KUKA KRL program: EPS_2_26115_SA7006_A_20260219035544.src

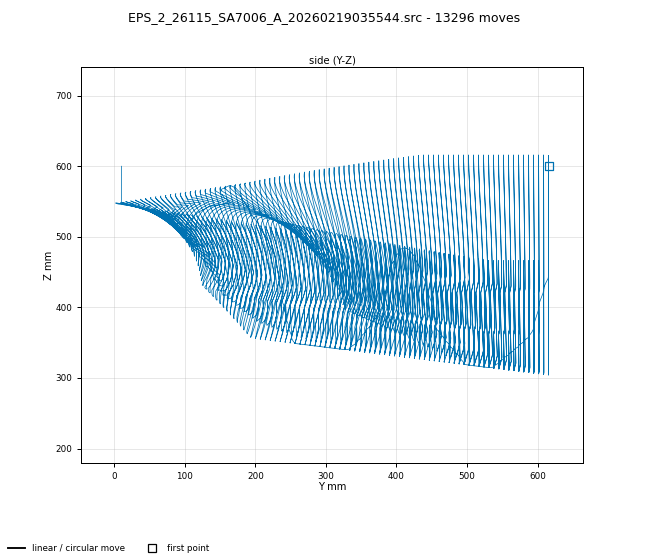
[picture p0: tool path of EPS_2_26115_SA7006_A_20260219035544.src, 13296 of 13298 moves have a stored position in this frame; points joined in program order, loops and branches not executed]
&ACCESS RVP
&REL 4
&COMMENT QRS 19112012
&PARAM EDITMASK = *
DEF PART()
EXT BAS (BAS_COMMAND :IN,REAL :IN )
INT I
BAS (#INITMOV,0 )

;KUKA QRS Post kuka4.cps  Date:22-06-2017 !

File_ID=3062

QRS_PRE_INIT()

;Init var - Until changes are made in qrs_pre_init
Outlet_Square_prg=0
Inlet_1_Square_prg=0
Inlet_2_Square_prg=0
Inlet_3_Square_prg=0
Inlet_4_Square_prg=0
Inlet_5_Square_prg=0

Outlet_1={X 0.000, Y 435.000, Z 433.000, B 0.000, E1 0.000 }
Inlet_1={X 0.000, Y 529.410, Z 340.500, B 0.000, E1 90.000 }
Inlet_2={X 0.000, Y 529.410, Z 340.500, B 0.000, E1 180.000 }
Outlet_1_type=366
Inlet_1_type=201
Inlet_2_type=201
;QRS#1=Sidecore dimensions
;QRS#2=375-15" PVC SDR 35 Cut Back
;QRS#3=200-8" PVC SDR 35
;QRS#4=200-8" PVC SDR 35
;QRS#5=
;QRS#6=
;QRS#7=
;QRS#8=
;QRS#9=20Y PSX
;QRS#10=12-08 PSX
;QRS#11=12-08 PSX
;QRS#12=
;QRS#13=
;QRS#14=
;QRS#15=
;QRS#16=1220x127x914 3'
;QRS#17=EPS Height
;QRS#18=616
;QRS#19=*
;QRS#20= UPDATED VERSION 22-06-2017
;QRS#21=*
Outlet_Square=0250
Inlet_1_Square=0100
Inlet_2_Square=0100
Inlet_3_Square=0
Inlet_4_Square=0
Inlet_5_Square=0
Mill_Square=1
Outlet_Square_Prg=275
Inlet_1_Square_prg=204
Inlet_2_Square_prg=204

QRS_INIT()

$ADVANCE=5

; T1
PTP {E1 173.498,E2 173.498}
PTP {X 0,Y 615.498,A -85,B 0,C 180,E1 173.498,E2 173.498,E3 0,E4 0,E5 0,E6 0}
QRS_SPEED_INIT()
LIN {X 0,Y 615.498,Z 600,A -85,B 0,C 180,E1 173.498,E2 173.498,E3 0,E4 0,E5 0,E6 0} C_VEL
LIN {X 0,Y 615.498,Z 456.733,A -85,B 0,C 180,E1 173.498,E2 173.498} C_VEL
LIN {X 0,Y 615.498,Z 445.854,A -85,B 0,C 180,E1 173.498,E2 173.498} C_VEL
LIN {X 0,Y 615.496,Z 444.21,A -85,B 0,C 180,E1 173.418,E2 173.418} C_VEL
LIN {X 0,Y 615.497,Z 436.534,A -85,B 0,C 180,E1 172.454,E2 172.454} C_VEL
LIN {X 0,Y 615.498,Z 426.756,A -85,B 0,C 180,E1 171.463,E2 171.463} C_VEL
LIN {X 0,Y 615.498,Z 416.489,A -85,B 0,C 180,E1 170.635,E2 170.635} C_VEL
LIN {X 0,Y 615.464,Z 404.93,A -85,B 0,C 180,E1 169.888,E2 169.888} C_VEL
LIN {X 0,Y 615.482,Z 393.083,A -85,B 0,C 180,E1 169.293,E2 169.293} C_VEL
LIN {X 0,Y 615.493,Z 380.15,A -85,B 0,C 180,E1 168.807,E2 168.807} C_VEL
LIN {X 0,Y 615.483,Z 367.548,A -85,B 0,C 180,E1 168.473,E2 168.473} C_VEL
LIN {X 0,Y 615.474,Z 360.281,A -85,B 0,C 180,E1 168.327,E2 168.327} C_VEL
LIN {X 0,Y 615.446,Z 354.613,A -85,B 0,C 180,E1 166.085,E2 166.085} C_VEL
LIN {X 0,Y 615.469,Z 347.897,A -85,B 0,C 180,E1 163.413,E2 163.413} C_VEL
LIN {X 0,Y 615.435,Z 341.109,A -85,B 0,C 180,E1 160.66,E2 160.66} C_VEL
LIN {X 0,Y 615.436,Z 335.997,A -85,B 0,C 180,E1 158.566,E2 158.566} C_VEL
LIN {X 0,Y 615.464,Z 329.821,A -85,B 0,C 180,E1 155.998,E2 155.998} C_VEL
LIN {X 0,Y 615.491,Z 324.07,A -85,B 0,C 180,E1 153.556,E2 153.556} C_VEL
LIN {X 0,Y 615.488,Z 318.958,A -85,B 0,C 180,E1 151.342,E2 151.342} C_VEL
LIN {X 0,Y 615.493,Z 313.469,A -85,B 0,C 180,E1 148.914,E2 148.914} C_VEL
LIN {X 0,Y 615.495,Z 307.987,A -85,B 0,C 180,E1 146.466,E2 146.466} C_VEL
LIN {X 0,Y 615.477,Z 304.012,A -85,B 0,C 180,E1 144.684,E2 144.684} C_VEL
LIN {X 0,Y 615.479,Z 304.01,A -85,B 0,C 180,E1 141.93,E2 141.93} C_VEL
LIN {X 0,Y 615.492,Z 304.007,A -85,B 0,C 180,E1 139.394,E2 139.394} C_VEL
LIN {X 0,Y 615.463,Z 304.012,A -85,B 0,C 180,E1 136.753,E2 136.753} C_VEL
LIN {X 0,Y 615.466,Z 304.012,A -85,B 0,C 180,E1 133.995,E2 133.995} C_VEL
LIN {X 0,Y 615.494,Z 304.011,A -85,B 0,C 180,E1 131.095,E2 131.095} C_VEL
LIN {X 0,Y 615.469,Z 304.011,A -85,B 0,C 180,E1 128.907,E2 128.907} C_VEL
LIN {X 0,Y 615.462,Z 304.013,A -85,B 0,C 180,E1 126.428,E2 126.428} C_VEL
LIN {X 0,Y 615.481,Z 304.167,A -85,B 0,C 180,E1 124.817,E2 124.817} C_VEL
LIN {X 0,Y 615.49,Z 310.295,A -85,B 0,C 180,E1 122.331,E2 122.331} C_VEL
LIN {X 0,Y 615.491,Z 316.167,A -85,B 0,C 180,E1 119.795,E2 119.795} C_VEL
LIN {X 0,Y 615.44,Z 322.494,A -85,B 0,C 180,E1 117.036,E2 117.036} C_VEL
LIN {X 0,Y 615.448,Z 327.267,A -85,B 0,C 180,E1 114.995,E2 114.995} C_VEL
LIN {X 0,Y 615.492,Z 333.562,A -85,B 0,C 180,E1 112.346,E2 112.346} C_VEL
LIN {X 0,Y 615.488,Z 339.166,A -85,B 0,C 180,E1 110.034,E2 110.034} C_VEL
LIN {X 0,Y 615.48,Z 345.979,A -85,B 0,C 180,E1 107.272,E2 107.272} C_VEL
LIN {X 0,Y 615.469,Z 352.77,A -85,B 0,C 180,E1 104.551,E2 104.551} C_VEL
LIN {X 0,Y 615.487,Z 359.577,A -85,B 0,C 180,E1 101.862,E2 101.862} C_VEL
LIN {X 0,Y 615.494,Z 360.311,A -85,B 0,C 180,E1 101.57,E2 101.57} C_VEL
LIN {X 0,Y 615.491,Z 372.644,A -85,B 0,C 180,E1 101.319,E2 101.319} C_VEL
LIN {X 0,Y 615.456,Z 385.792,A -85,B 0,C 180,E1 100.911,E2 100.911} C_VEL
LIN {X 0,Y 615.455,Z 398.542,A -85,B 0,C 180,E1 100.363,E2 100.363} C_VEL
LIN {X 0,Y 615.497,Z 410.282,A -85,B 0,C 180,E1 99.697,E2 99.697} C_VEL
LIN {X 0,Y 615.499,Z 420.75,A -85,B 0,C 180,E1 98.952,E2 98.952} C_VEL
LIN {X 0,Y 615.498,Z 429.315,A -85,B 0,C 180,E1 98.207,E2 98.207} C_VEL
LIN {X 0,Y 615.497,Z 437.196,A -85,B 0,C 180,E1 97.382,E2 97.382} C_VEL
LIN {X 0,Y 615.497,Z 444.889,A -85,B 0,C 180,E1 96.393,E2 96.393} C_VEL
LIN {X 0,Y 615.497,Z 451.95,A -85,B 0,C 180,E1 95.243,E2 95.243} C_VEL
LIN {X 0,Y 615.494,Z 456.651,A -85,B 0,C 180,E1 94.258,E2 94.258} C_VEL
LIN {X 0,Y 615.494,Z 460.25,A -85,B 0,C 180,E1 93.274,E2 93.274} C_VEL
LIN {X 0,Y 615.496,Z 462.111,A -85,B 0,C 180,E1 92.619,E2 92.619} C_VEL
LIN {X 0,Y 615.499,Z 463.53,A -85,B 0,C 180,E1 91.965,E2 91.965} C_VEL
LIN {X 0,Y 615.496,Z 465.14,A -85,B 0,C 180,E1 90.656,E2 90.656} C_VEL
LIN {X 0,Y 615.495,Z 465.384,A -85,B 0,C 180,E1 90.002,E2 90.002} C_VEL
LIN {X 0,Y 615.495,Z 465.207,A -85,B 0,C 180,E1 89.347,E2 89.347} C_VEL
LIN {X 0,Y 615.499,Z 463.685,A -85,B 0,C 180,E1 88.039,E2 88.039} C_VEL
LIN {X 0,Y 615.498,Z 462.345,A -85,B 0,C 180,E1 87.384,E2 87.384} C_VEL
LIN {X 0,Y 615.496,Z 459.499,A -85,B 0,C 180,E1 86.401,E2 86.401} C_VEL
LIN {X 0,Y 615.498,Z 455.641,A -85,B 0,C 180,E1 85.417,E2 85.417} C_VEL
LIN {X 0,Y 615.498,Z 450.661,A -85,B 0,C 180,E1 84.432,E2 84.432} C_VEL
LIN {X 0,Y 615.496,Z 444.209,A -85,B 0,C 180,E1 83.418,E2 83.418} C_VEL
LIN {X 0,Y 615.497,Z 436.553,A -85,B 0,C 180,E1 82.456,E2 82.456} C_VEL
LIN {X 0,Y 615.498,Z 426.778,A -85,B 0,C 180,E1 81.465,E2 81.465} C_VEL
LIN {X 0,Y 615.498,Z 416.518,A -85,B 0,C 180,E1 80.637,E2 80.637} C_VEL
LIN {X 0,Y 615.472,Z 404.964,A -85,B 0,C 180,E1 79.89,E2 79.89} C_VEL
LIN {X 0,Y 615.444,Z 393.348,A -85,B 0,C 180,E1 79.303,E2 79.303} C_VEL
LIN {X 0,Y 615.466,Z 381.479,A -85,B 0,C 180,E1 78.849,E2 78.849} C_VEL
LIN {X 0,Y 615.491,Z 369.465,A -85,B 0,C 180,E1 78.517,E2 78.517} C_VEL
LIN {X 0,Y 615.495,Z 360.283,A -85,B 0,C 180,E1 78.329,E2 78.329} C_VEL
LIN {X 0,Y 615.49,Z 354.559,A -85,B 0,C 180,E1 76.068,E2 76.068} C_VEL
LIN {X 0,Y 615.472,Z 347.903,A -85,B 0,C 180,E1 73.415,E2 73.415} C_VEL
LIN {X 0,Y 615.476,Z 341.109,A -85,B 0,C 180,E1 70.664,E2 70.664} C_VEL
LIN {X 0,Y 615.488,Z 334.288,A -85,B 0,C 180,E1 67.866,E2 67.866} C_VEL
LIN {X 0,Y 615.489,Z 329.182,A -85,B 0,C 180,E1 65.73,E2 65.73} C_VEL
LIN {X 0,Y 615.467,Z 324.079,A -85,B 0,C 180,E1 63.557,E2 63.557} C_VEL
LIN {X 0,Y 615.437,Z 318.971,A -85,B 0,C 180,E1 61.342,E2 61.342} C_VEL
LIN {X 0,Y 615.489,Z 313.418,A -85,B 0,C 180,E1 58.914,E2 58.914} C_VEL
LIN {X 0,Y 615.499,Z 307.609,A -85,B 0,C 180,E1 56.465,E2 56.465} C_VEL
LIN {X 0,Y 615.481,Z 304.007,A -85,B 0,C 180,E1 54.988,E2 54.988} C_VEL
LIN {X 0,Y 615.475,Z 304.002,A -85,B 0,C 180,E1 52.76,E2 52.76} C_VEL
LIN {X 0,Y 615.48,Z 304.012,A -85,B 0,C 180,E1 49.912,E2 49.912} C_VEL
LIN {X 0,Y 615.433,Z 304.012,A -85,B 0,C 180,E1 47.646,E2 47.646} C_VEL
LIN {X 0,Y 615.48,Z 304.013,A -85,B 0,C 180,E1 44.934,E2 44.934} C_VEL
LIN {X 0,Y 615.468,Z 304.004,A -85,B 0,C 180,E1 42.082,E2 42.082} C_VEL
LIN {X 0,Y 615.487,Z 304.01,A -85,B 0,C 180,E1 39.751,E2 39.751} C_VEL
LIN {X 0,Y 615.471,Z 304.003,A -85,B 0,C 180,E1 36.939,E2 36.939} C_VEL
LIN {X 0,Y 615.46,Z 304.012,A -85,B 0,C 180,E1 34.024,E2 34.024} C_VEL
LIN {X 0,Y 615.429,Z 304.012,A -85,B 0,C 180,E1 31.689,E2 31.689} C_VEL
LIN {X 0,Y 615.463,Z 304.012,A -85,B 0,C 180,E1 29.408,E2 29.408} C_VEL
LIN {X 0,Y 615.477,Z 304.002,A -85,B 0,C 180,E1 26.445,E2 26.445} C_VEL
LIN {X 0,Y 615.483,Z 304.011,A -85,B 0,C 180,E1 24.014,E2 24.014} C_VEL
LIN {X 0,Y 615.458,Z 304.007,A -85,B 0,C 180,E1 21.433,E2 21.433} C_VEL
LIN {X 0,Y 615.49,Z 304.015,A -85,B 0,C 180,E1 18.614,E2 18.614} C_VEL
LIN {X 0,Y 615.432,Z 304.012,A -85,B 0,C 180,E1 15.907,E2 15.907} C_VEL
LIN {X 0,Y 615.495,Z 304.008,A -85,B 0,C 180,E1 13.201,E2 13.201} C_VEL
LIN {X 0,Y 615.477,Z 304.003,A -85,B 0,C 180,E1 10.527,E2 10.527} C_VEL
LIN {X 0,Y 615.478,Z 304.01,A -85,B 0,C 180,E1 7.876,E2 7.876} C_VEL
LIN {X 0,Y 615.469,Z 304.005,A -85,B 0,C 180,E1 5.242,E2 5.242} C_VEL
LIN {X 0,Y 615.463,Z 304.012,A -85,B 0,C 180,E1 2.618,E2 2.618} C_VEL
LIN {X 0,Y 615.444,Z 304.011,A -85,B 0,C 180,E1 0,E2 0} C_VEL
LIN {X 0,Y 615.491,Z 304.006,A -85,B 0,C 180,E1 -2.618,E2 -2.618} C_VEL
LIN {X 0,Y 615.481,Z 304.002,A -85,B 0,C 180,E1 -5.241,E2 -5.241} C_VEL
LIN {X 0,Y 615.473,Z 304.01,A -85,B 0,C 180,E1 -7.876,E2 -7.876} C_VEL
LIN {X 0,Y 615.461,Z 304.007,A -85,B 0,C 180,E1 -10.527,E2 -10.527} C_VEL
LIN {X 0,Y 615.456,Z 304.012,A -85,B 0,C 180,E1 -13.202,E2 -13.202} C_VEL
LIN {X 0,Y 615.46,Z 304.007,A -85,B 0,C 180,E1 -15.226,E2 -15.226} C_VEL
LIN {X 0,Y 615.484,Z 304.012,A -85,B 0,C 180,E1 -17.957,E2 -17.957} C_VEL
LIN {X 0,Y 615.492,Z 303.998,A -85,B 0,C 180,E1 -20.73,E2 -20.73} C_VEL
LIN {X 0,Y 615.474,Z 304.011,A -85,B 0,C 180,E1 -23.557,E2 -23.557} C_VEL
LIN {X 0,Y 615.437,Z 304.012,A -85,B 0,C 180,E1 -25.718,E2 -25.718} C_VEL
LIN {X 0,Y 615.481,Z 304.013,A -85,B 0,C 180,E1 -28.455,E2 -28.455} C_VEL
LIN {X 0,Y 615.462,Z 304.005,A -85,B 0,C 180,E1 -31.087,E2 -31.087} C_VEL
LIN {X 0,Y 615.478,Z 304.009,A -85,B 0,C 180,E1 -33.538,E2 -33.538} C_VEL
LIN {X 0,Y 615.481,Z 304.001,A -85,B 0,C 180,E1 -36.425,E2 -36.425} C_VEL
LIN {X 0,Y 615.492,Z 304.014,A -85,B 0,C 180,E1 -39.067,E2 -39.067} C_VEL
LIN {X 0,Y 615.433,Z 304.012,A -85,B 0,C 180,E1 -41.478,E2 -41.478} C_VEL
LIN {X 0,Y 615.48,Z 304.013,A -85,B 0,C 180,E1 -44.15,E2 -44.15} C_VEL
LIN {X 0,Y 615.464,Z 304.005,A -85,B 0,C 180,E1 -46.955,E2 -46.955} C_VEL
LIN {X 0,Y 615.489,Z 304.011,A -85,B 0,C 180,E1 -49.397,E2 -49.397} C_VEL
LIN {X 0,Y 615.471,Z 304.003,A -85,B 0,C 180,E1 -51.99,E2 -51.99} C_VEL
LIN {X 0,Y 615.497,Z 304.002,A -85,B 0,C 180,E1 -54.388,E2 -54.388} C_VEL
LIN {X 0,Y 615.444,Z 304.194,A -85,B 0,C 180,E1 -55.768,E2 -55.768} C_VEL
LIN {X 0,Y 615.497,Z 324.712,A -85,B 0,C 180,E1 -58.468,E2 -58.468} C_VEL
LIN {X 0,Y 615.482,Z 347.265,A -85,B 0,C 180,E1 -61.344,E2 -61.344} C_VEL
LIN {X 0,Y 615.489,Z 369.495,A -85,B 0,C 180,E1 -64.105,E2 -64.105} C_VEL
LIN {X 0,Y 615.479,Z 391.725,A -85,B 0,C 180,E1 -66.802,E2 -66.802} C_VEL
LIN {X 0,Y 615.491,Z 415.039,A -85,B 0,C 180,E1 -69.574,E2 -69.574} C_VEL
LIN {X 0,Y 615.494,Z 421.023,A -85,B 0,C 180,E1 -70.252,E2 -70.252} C_VEL
LIN {X 0,Y 615.487,Z 444.892,A -85,B 0,C 180,E1 -70.578,E2 -70.578} C_VEL
LIN {X 0,Y 615.475,Z 460.906,A -85,B 0,C 180,E1 -70.924,E2 -70.924} C_VEL
LIN {X 0,Y 615.493,Z 476.391,A -85,B 0,C 180,E1 -71.393,E2 -71.393} C_VEL
LIN {X 0,Y 615.488,Z 491.252,A -85,B 0,C 180,E1 -71.964,E2 -71.964} C_VEL
LIN {X 0,Y 615.499,Z 505.771,A -85,B 0,C 180,E1 -72.646,E2 -72.646} C_VEL
LIN {X 0,Y 615.498,Z 520.515,A -85,B 0,C 180,E1 -73.49,E2 -73.49} C_VEL
LIN {X 0,Y 615.497,Z 534.385,A -85,B 0,C 180,E1 -74.437,E2 -74.437} C_VEL
LIN {X 0,Y 615.495,Z 547.051,A -85,B 0,C 180,E1 -75.453,E2 -75.453} C_VEL
LIN {X 0,Y 615.493,Z 559.563,A -85,B 0,C 180,E1 -76.633,E2 -76.633} C_VEL
LIN {X 0,Y 615.49,Z 570.189,A -85,B 0,C 180,E1 -77.807,E2 -77.807} C_VEL
LIN {X 0,Y 615.49,Z 580.236,A -85,B 0,C 180,E1 -79.11,E2 -79.11} C_VEL
LIN {X 0,Y 615.495,Z 588.995,A -85,B 0,C 180,E1 -80.472,E2 -80.472} C_VEL
LIN {X 0,Y 615.495,Z 596.117,A -85,B 0,C 180,E1 -81.796,E2 -81.796} C_VEL
LIN {X 0,Y 615.491,Z 601.986,A -85,B 0,C 180,E1 -83.103,E2 -83.103} C_VEL
LIN {X 0,Y 615.492,Z 607.746,A -85,B 0,C 180,E1 -84.761,E2 -84.761} C_VEL
LIN {X 0,Y 615.493,Z 611.08,A -85,B 0,C 180,E1 -86.073,E2 -86.073} C_VEL
LIN {X 0,Y 615.485,Z 613.507,A -85,B 0,C 180,E1 -87.384,E2 -87.384} C_VEL
LIN {X 0,Y 615.488,Z 614.871,A -85,B 0,C 180,E1 -88.693,E2 -88.693} C_VEL
LIN {X 0,Y 615.489,Z 615.39,A -85,B 0,C 180,E1 -90.002,E2 -90.002} C_VEL
LIN {X 0,Y 615.488,Z 614.869,A -85,B 0,C 180,E1 -91.31,E2 -91.31} C_VEL
LIN {X 0,Y 615.485,Z 613.502,A -85,B 0,C 180,E1 -92.619,E2 -92.619} C_VEL
LIN {X 0,Y 615.493,Z 611.073,A -85,B 0,C 180,E1 -93.93,E2 -93.93} C_VEL
LIN {X 0,Y 615.492,Z 607.736,A -85,B 0,C 180,E1 -95.243,E2 -95.243} C_VEL
LIN {X 0,Y 615.492,Z 601.979,A -85,B 0,C 180,E1 -96.899,E2 -96.899} C_VEL
LIN {X 0,Y 615.489,Z 594.494,A -85,B 0,C 180,E1 -98.538,E2 -98.538} C_VEL
LIN {X 0,Y 615.496,Z 585.955,A -85,B 0,C 180,E1 -100.029,E2 -100.029} C_VEL
LIN {X 0,Y 615.494,Z 576.756,A -85,B 0,C 180,E1 -101.361,E2 -101.361} C_VEL
LIN {X 0,Y 615.495,Z 567.279,A -85,B 0,C 180,E1 -102.531,E2 -102.531} C_VEL
LIN {X 0,Y 615.496,Z 556.199,A -85,B 0,C 180,E1 -103.707,E2 -103.707} C_VEL
LIN {X 0,Y 615.495,Z 544.099,A -85,B 0,C 180,E1 -104.804,E2 -104.804} C_VEL
LIN {X 0,Y 615.497,Z 529.69,A -85,B 0,C 180,E1 -105.906,E2 -105.906} C_VEL
LIN {X 0,Y 615.497,Z 514.993,A -85,B 0,C 180,E1 -106.844,E2 -106.844} C_VEL
LIN {X 0,Y 615.499,Z 500.484,A -85,B 0,C 180,E1 -107.614,E2 -107.614} C_VEL
LIN {X 0,Y 615.486,Z 485.241,A -85,B 0,C 180,E1 -108.282,E2 -108.282} C_VEL
LIN {X 0,Y 615.48,Z 469.949,A -85,B 0,C 180,E1 -108.82,E2 -108.82} C_VEL
LIN {X 0,Y 615.478,Z 453.466,A -85,B 0,C 180,E1 -109.253,E2 -109.253} C_VEL
LIN {X 0,Y 615.494,Z 437.841,A -85,B 0,C 180,E1 -109.534,E2 -109.534} C_VEL
LIN {X 0,Y 615.494,Z 420.778,A -85,B 0,C 180,E1 -109.751,E2 -109.751} C_VEL
LIN {X 0,Y 615.496,Z 396.751,A -85,B 0,C 180,E1 -112.595,E2 -112.595} C_VEL
LIN {X 0,Y 615.489,Z 373.317,A -85,B 0,C 180,E1 -115.427,E2 -115.427} C_VEL
LIN {X 0,Y 615.488,Z 349.955,A -85,B 0,C 180,E1 -118.318,E2 -118.318} C_VEL
LIN {X 0,Y 615.474,Z 328.189,A -85,B 0,C 180,E1 -121.084,E2 -121.084} C_VEL
LIN {X 0,Y 615.485,Z 307.571,A -85,B 0,C 180,E1 -123.78,E2 -123.78} C_VEL
LIN {X 0,Y 615.464,Z 304.011,A -85,B 0,C 180,E1 -124.278,E2 -124.278} C_VEL
LIN {X 0,Y 615.483,Z 304.012,A -85,B 0,C 180,E1 -126.426,E2 -126.426} C_VEL
LIN {X 0,Y 615.494,Z 304.013,A -85,B 0,C 180,E1 -129.063,E2 -129.063} C_VEL
LIN {X 0,Y 615.491,Z 304.007,A -85,B 0,C 180,E1 -131.475,E2 -131.475} C_VEL
LIN {X 0,Y 615.473,Z 304.01,A -85,B 0,C 180,E1 -134.152,E2 -134.152} C_VEL
LIN {X 0,Y 615.456,Z 304.012,A -85,B 0,C 180,E1 -136.753,E2 -136.753} C_VEL
LIN {X 0,Y 615.494,Z 304.004,A -85,B 0,C 180,E1 -139.394,E2 -139.394} C_VEL
LIN {X 0,Y 615.461,Z 304.013,A -85,B 0,C 180,E1 -141.992,E2 -141.992} C_VEL
LIN {X 0,Y 615.495,Z 304.012,A -85,B 0,C 180,E1 -144.385,E2 -144.385} C_VEL
LIN {X 0,Y 615.498,Z 304.193,A -85,B 0,C 180,E1 -145.471,E2 -145.471} C_VEL
LIN {X 0,Y 615.489,Z 310.175,A -85,B 0,C 180,E1 -147.67,E2 -147.67} C_VEL
LIN {X 0,Y 615.494,Z 316.167,A -85,B 0,C 180,E1 -150.205,E2 -150.205} C_VEL
LIN {X 0,Y 615.473,Z 322.473,A -85,B 0,C 180,E1 -152.959,E2 -152.959} C_VEL
LIN {X 0,Y 615.49,Z 328.964,A -85,B 0,C 180,E1 -155.728,E2 -155.728} C_VEL
LIN {X 0,Y 615.468,Z 334.07,A -85,B 0,C 180,E1 -157.863,E2 -157.863} C_VEL
LIN {X 0,Y 615.441,Z 339.177,A -85,B 0,C 180,E1 -159.966,E2 -159.966} C_VEL
LIN {X 0,Y 615.424,Z 344.283,A -85,B 0,C 180,E1 -162.041,E2 -162.041} C_VEL
LIN {X 0,Y 615.471,Z 351.079,A -85,B 0,C 180,E1 -164.774,E2 -164.774} C_VEL
LIN {X 0,Y 615.464,Z 357.873,A -85,B 0,C 180,E1 -167.47,E2 -167.47} C_VEL
LIN {X 0,Y 615.474,Z 360.319,A -85,B 0,C 180,E1 -168.432,E2 -168.432} C_VEL
LIN {X 0,Y 615.495,Z 372.705,A -85,B 0,C 180,E1 -168.682,E2 -168.682} C_VEL
LIN {X 0,Y 615.486,Z 385.417,A -85,B 0,C 180,E1 -169.076,E2 -169.076} C_VEL
LIN {X 0,Y 615.462,Z 396.832,A -85,B 0,C 180,E1 -169.556,E2 -169.556} C_VEL
LIN {X 0,Y 615.467,Z 407.633,A -85,B 0,C 180,E1 -170.138,E2 -170.138} C_VEL
LIN {X 0,Y 615.498,Z 418.662,A -85,B 0,C 180,E1 -170.884,E2 -170.884} C_VEL
LIN {X 0,Y 615.498,Z 429.333,A -85,B 0,C 180,E1 -171.794,E2 -171.794} C_VEL
LIN {X 0,Y 615.497,Z 437.211,A -85,B 0,C 180,E1 -172.62,E2 -172.62} C_VEL
LIN {X 0,Y 615.497,Z 444.9,A -85,B 0,C 180,E1 -173.608,E2 -173.608} C_VEL
LIN {X 0,Y 615.497,Z 451.959,A -85,B 0,C 180,E1 -174.759,E2 -174.759} C_VEL
LIN {X 0,Y 615.493,Z 456.659,A -85,B 0,C 180,E1 -175.744,E2 -175.744} C_VEL
LIN {X 0,Y 615.495,Z 460.255,A -85,B 0,C 180,E1 -176.727,E2 -176.727} C_VEL
LIN {X 0,Y 615.496,Z 462.115,A -85,B 0,C 180,E1 -177.382,E2 -177.382} C_VEL
LIN {X 0,Y 615.497,Z 463.534,A -85,B 0,C 180,E1 -178.037,E2 -178.037} C_VEL
LIN {X 0,Y 615.496,Z 465.142,A -85,B 0,C 180,E1 -179.346,E2 -179.346} C_VEL
LIN {X 0,Y 615.494,Z 465.384,A -85,B 0,C 180,E1 -180,E2 -180} C_VEL
LIN {X 0,Y 615.495,Z 465.205,A -85,B 0,C 180,E1 -180.654,E2 -180.654} C_VEL
LIN {X 0,Y 615.496,Z 463.683,A -85,B 0,C 180,E1 -181.963,E2 -181.963} C_VEL
LIN {X 0,Y 615.498,Z 462.341,A -85,B 0,C 180,E1 -182.618,E2 -182.618} C_VEL
LIN {X 0,Y 615.496,Z 459.493,A -85,B 0,C 180,E1 -183.601,E2 -183.601} C_VEL
LIN {X 0,Y 615.498,Z 455.633,A -85,B 0,C 180,E1 -184.585,E2 -184.585} C_VEL
LIN {X 0,Y 615.498,Z 450.65,A -85,B 0,C 180,E1 -185.57,E2 -185.57} C_VEL
LIN {X 0,Y 615.496,Z 444.21,A -85,B 0,C 180,E1 -186.582,E2 -186.582} C_VEL
LIN {X 0,Y 614.829,Z 441.028,A -85,B 0,C 180,E1 -187.031,E2 -187.031} C_VEL
LIN {X 0,Y 611.989,Z 435.455,A -85,B 0,C 180,E1 -187.748,E2 -187.748} C_VEL
LIN {X 0,Y 609.138,Z 429.18,A -85,B 0,C 180,E1 -188.429,E2 -188.429} C_VEL
LIN {X 0,Y 608.477,Z 424.939,A -85,B 0,C 180,E1 -188.819,E2 -188.819} C_VEL
LIN {X 0,Y 608.49,Z 414.386,A -85,B 0,C 180,E1 -189.641,E2 -189.641} C_VEL
LIN {X 0,Y 608.465,Z 403.606,A -85,B 0,C 180,E1 -190.314,E2 -190.314} C_VEL
LIN {X 0,Y 608.527,Z 391.967,A -85,B 0,C 180,E1 -190.884,E2 -190.884} C_VEL
LIN {X 0,Y 608.539,Z 378.958,A -85,B 0,C 180,E1 -191.365,E2 -191.365} C_VEL
LIN {X 0,Y 608.537,Z 366.644,A -85,B 0,C 180,E1 -191.682,E2 -191.682} C_VEL
LIN {X 0,Y 608.428,Z 360.677,A -85,B 0,C 180,E1 -191.81,E2 -191.81} C_VEL
LIN {X 0,Y 608.429,Z 353.349,A -85,B 0,C 180,E1 -194.722,E2 -194.722} C_VEL
LIN {X 0,Y 608.396,Z 346.502,A -85,B 0,C 180,E1 -197.479,E2 -197.479} C_VEL
LIN {X 0,Y 608.385,Z 341.367,A -85,B 0,C 180,E1 -199.573,E2 -199.573} C_VEL
LIN {X 0,Y 608.406,Z 336.231,A -85,B 0,C 180,E1 -201.694,E2 -201.694} C_VEL
LIN {X 0,Y 608.442,Z 330.393,A -85,B 0,C 180,E1 -204.144,E2 -204.144} C_VEL
LIN {X 0,Y 608.433,Z 324.248,A -85,B 0,C 180,E1 -206.775,E2 -206.775} C_VEL
LIN {X 0,Y 608.434,Z 319.112,A -85,B 0,C 180,E1 -209.022,E2 -209.022} C_VEL
LIN {X 0,Y 608.484,Z 313.982,A -85,B 0,C 180,E1 -211.316,E2 -211.316} C_VEL
LIN {X 0,Y 608.479,Z 308.591,A -85,B 0,C 180,E1 -213.735,E2 -213.735} C_VEL
LIN {X 0,Y 608.458,Z 305.007,A -85,B 0,C 180,E1 -215.378,E2 -215.378} C_VEL
LIN {X 0,Y 608.465,Z 305.005,A -85,B 0,C 180,E1 -218.239,E2 -218.239} C_VEL
LIN {X 0,Y 608.465,Z 305.008,A -85,B 0,C 180,E1 -221.342,E2 -221.342} C_VEL
LIN {X 0,Y 608.463,Z 305.006,A -85,B 0,C 180,E1 -224.263,E2 -224.263} C_VEL
LIN {X 0,Y 608.435,Z 305.009,A -85,B 0,C 180,E1 -227.038,E2 -227.038} C_VEL
LIN {X 0,Y 608.461,Z 305.005,A -85,B 0,C 180,E1 -229.696,E2 -229.696} C_VEL
LIN {X 0,Y 608.48,Z 305.007,A -85,B 0,C 180,E1 -232.841,E2 -232.841} C_VEL
LIN {X 0,Y 608.476,Z 305.008,A -85,B 0,C 180,E1 -235.091,E2 -235.091} C_VEL
LIN {X 0,Y 608.463,Z 310.869,A -85,B 0,C 180,E1 -237.478,E2 -237.478} C_VEL
LIN {X 0,Y 608.476,Z 317.184,A -85,B 0,C 180,E1 -240.22,E2 -240.22} C_VEL
LIN {X 0,Y 608.4,Z 324.038,A -85,B 0,C 180,E1 -243.222,E2 -243.222} C_VEL
LIN {X 0,Y 608.44,Z 329.17,A -85,B 0,C 180,E1 -245.427,E2 -245.427} C_VEL
LIN {X 0,Y 608.437,Z 336.013,A -85,B 0,C 180,E1 -248.306,E2 -248.306} C_VEL
LIN {X 0,Y 608.434,Z 342.856,A -85,B 0,C 180,E1 -251.128,E2 -251.128} C_VEL
LIN {X 0,Y 608.441,Z 349.699,A -85,B 0,C 180,E1 -253.904,E2 -253.904} C_VEL
LIN {X 0,Y 608.438,Z 356.543,A -85,B 0,C 180,E1 -256.642,E2 -256.642} C_VEL
LIN {X 0,Y 608.448,Z 360.714,A -85,B 0,C 180,E1 -258.294,E2 -258.294} C_VEL
LIN {X 0,Y 608.535,Z 374.311,A -85,B 0,C 180,E1 -258.592,E2 -258.592} C_VEL
LIN {X 0,Y 608.491,Z 387.182,A -85,B 0,C 180,E1 -259.01,E2 -259.01} C_VEL
LIN {X 0,Y 608.472,Z 398.709,A -85,B 0,C 180,E1 -259.517,E2 -259.517} C_VEL
LIN {X 0,Y 608.487,Z 410.487,A -85,B 0,C 180,E1 -260.19,E2 -260.19} C_VEL
LIN {X 0,Y 608.485,Z 421.005,A -85,B 0,C 180,E1 -260.944,E2 -260.944} C_VEL
LIN {X 0,Y 608.476,Z 429.618,A -85,B 0,C 180,E1 -261.697,E2 -261.697} C_VEL
LIN {X 0,Y 608.471,Z 437.551,A -85,B 0,C 180,E1 -262.532,E2 -262.532} C_VEL
LIN {X 0,Y 608.469,Z 445.065,A -85,B 0,C 180,E1 -263.497,E2 -263.497} C_VEL
LIN {X 0,Y 608.451,Z 450.601,A -85,B 0,C 180,E1 -264.364,E2 -264.364} C_VEL
LIN {X 0,Y 608.431,Z 455.744,A -85,B 0,C 180,E1 -265.361,E2 -265.361} C_VEL
LIN {X 0,Y 608.449,Z 459.735,A -85,B 0,C 180,E1 -266.356,E2 -266.356} C_VEL
LIN {X 0,Y 608.425,Z 462.687,A -85,B 0,C 180,E1 -267.35,E2 -267.35} C_VEL
LIN {X 0,Y 608.444,Z 464.124,A -85,B 0,C 180,E1 -268.013,E2 -268.013} C_VEL
LIN {X 0,Y 608.439,Z 465.751,A -85,B 0,C 180,E1 -269.337,E2 -269.337} C_VEL
LIN {X 0,Y 608.435,Z 465.995,A -85,B 0,C 180,E1 -269.998,E2 -269.998} C_VEL
LIN {X 0,Y 608.438,Z 465.816,A -85,B 0,C 180,E1 -270.66,E2 -270.66} C_VEL
LIN {X 0,Y 608.444,Z 464.279,A -85,B 0,C 180,E1 -271.984,E2 -271.984} C_VEL
LIN {X 0,Y 608.426,Z 462.921,A -85,B 0,C 180,E1 -272.647,E2 -272.647} C_VEL
LIN {X 0,Y 608.449,Z 460.046,A -85,B 0,C 180,E1 -273.641,E2 -273.641} C_VEL
LIN {X 0,Y 608.433,Z 456.148,A -85,B 0,C 180,E1 -274.636,E2 -274.636} C_VEL
LIN {X 0,Y 608.45,Z 451.12,A -85,B 0,C 180,E1 -275.633,E2 -275.633} C_VEL
LIN {X 0,Y 608.441,Z 444.807,A -85,B 0,C 180,E1 -276.631,E2 -276.631} C_VEL
LIN {X 0,Y 608.475,Z 436.894,A -85,B 0,C 180,E1 -277.631,E2 -277.631} C_VEL
LIN {X 0,Y 608.472,Z 427.051,A -85,B 0,C 180,E1 -278.634,E2 -278.634} C_VEL
LIN {X 0,Y 608.481,Z 416.74,A -85,B 0,C 180,E1 -279.471,E2 -279.471} C_VEL
LIN {X 0,Y 608.482,Z 405.133,A -85,B 0,C 180,E1 -280.227,E2 -280.227} C_VEL
LIN {X 0,Y 608.465,Z 393.459,A -85,B 0,C 180,E1 -280.821,E2 -280.821} C_VEL
LIN {X 0,Y 608.496,Z 381.359,A -85,B 0,C 180,E1 -281.287,E2 -281.287} C_VEL
LIN {X 0,Y 608.534,Z 368.637,A -85,B 0,C 180,E1 -281.637,E2 -281.637} C_VEL
LIN {X 0,Y 608.45,Z 360.682,A -85,B 0,C 180,E1 -281.808,E2 -281.808} C_VEL
LIN {X 0,Y 608.429,Z 353.355,A -85,B 0,C 180,E1 -284.72,E2 -284.72} C_VEL
LIN {X 0,Y 608.433,Z 346.508,A -85,B 0,C 180,E1 -287.475,E2 -287.475} C_VEL
LIN {X 0,Y 608.444,Z 339.661,A -85,B 0,C 180,E1 -290.273,E2 -290.273} C_VEL
LIN {X 0,Y 608.44,Z 332.814,A -85,B 0,C 180,E1 -293.122,E2 -293.122} C_VEL
LIN {X 0,Y 608.44,Z 325.966,A -85,B 0,C 180,E1 -296.033,E2 -296.033} C_VEL
LIN {X 0,Y 608.404,Z 320.055,A -85,B 0,C 180,E1 -298.607,E2 -298.607} C_VEL
LIN {X 0,Y 608.443,Z 315.674,A -85,B 0,C 180,E1 -300.544,E2 -300.544} C_VEL
LIN {X 0,Y 608.459,Z 310.262,A -85,B 0,C 180,E1 -302.877,E2 -302.877} C_VEL
LIN {X 0,Y 608.452,Z 305.006,A -85,B 0,C 180,E1 -305.06,E2 -305.06} C_VEL
LIN {X 0,Y 608.469,Z 305.002,A -85,B 0,C 180,E1 -307.743,E2 -307.743} C_VEL
LIN {X 0,Y 608.428,Z 305.008,A -85,B 0,C 180,E1 -310.326,E2 -310.326} C_VEL
LIN {X 0,Y 608.459,Z 305.008,A -85,B 0,C 180,E1 -313.307,E2 -313.307} C_VEL
LIN {X 0,Y 608.442,Z 305.004,A -85,B 0,C 180,E1 -316.128,E2 -316.128} C_VEL
LIN {X 0,Y 608.456,Z 305.008,A -85,B 0,C 180,E1 -318.823,E2 -318.823} C_VEL
LIN {X 0,Y 608.462,Z 305.003,A -85,B 0,C 180,E1 -321.756,E2 -321.756} C_VEL
LIN {X 0,Y 608.462,Z 305.009,A -85,B 0,C 180,E1 -323.948,E2 -323.948} C_VEL
LIN {X 0,Y 608.421,Z 305.007,A -85,B 0,C 180,E1 -326.326,E2 -326.326} C_VEL
LIN {X 0,Y 608.423,Z 305.008,A -85,B 0,C 180,E1 -328.731,E2 -328.731} C_VEL
LIN {X 0,Y 608.467,Z 305.002,A -85,B 0,C 180,E1 -331.375,E2 -331.375} C_VEL
LIN {X 0,Y 608.441,Z 305.006,A -85,B 0,C 180,E1 -333.964,E2 -333.964} C_VEL
LIN {X 0,Y 608.461,Z 305.01,A -85,B 0,C 180,E1 -336.155,E2 -336.155} C_VEL
LIN {X 0,Y 608.455,Z 305.004,A -85,B 0,C 180,E1 -338.308,E2 -338.308} C_VEL
LIN {X 0,Y 608.463,Z 305.008,A -85,B 0,C 180,E1 -341.277,E2 -341.277} C_VEL
LIN {X 0,Y 608.416,Z 305.007,A -85,B 0,C 180,E1 -343.905,E2 -343.905} C_VEL
LIN {X 0,Y 608.461,Z 305.01,A -85,B 0,C 180,E1 -346.643,E2 -346.643} C_VEL
LIN {X 0,Y 608.458,Z 305.002,A -85,B 0,C 180,E1 -349.35,E2 -349.35} C_VEL
LIN {X 0,Y 608.467,Z 305.006,A -85,B 0,C 180,E1 -352.033,E2 -352.033} C_VEL
LIN {X 0,Y 608.446,Z 305.003,A -85,B 0,C 180,E1 -354.698,E2 -354.698} C_VEL
LIN {X 0,Y 608.454,Z 305.007,A -85,B 0,C 180,E1 -357.352,E2 -357.352} C_VEL
LIN {X 0,Y 608.437,Z 305.005,A -85,B 0,C 180,E1 -360,E2 -360} C_VEL
LIN {X 0,Y 608.479,Z 305.003,A -85,B 0,C 180,E1 -362.648,E2 -362.648} C_VEL
LIN {X 0,Y 608.461,Z 305.002,A -85,B 0,C 180,E1 -365.302,E2 -365.302} C_VEL
LIN {X 0,Y 608.461,Z 305.004,A -85,B 0,C 180,E1 -367.967,E2 -367.967} C_VEL
LIN {X 0,Y 608.449,Z 305.005,A -85,B 0,C 180,E1 -370.65,E2 -370.65} C_VEL
LIN {X 0,Y 608.428,Z 305.007,A -85,B 0,C 180,E1 -373.357,E2 -373.357} C_VEL
LIN {X 0,Y 608.443,Z 305.003,A -85,B 0,C 180,E1 -375.406,E2 -375.406} C_VEL
LIN {X 0,Y 608.449,Z 305.01,A -85,B 0,C 180,E1 -378.172,E2 -378.172} C_VEL
LIN {X 0,Y 608.455,Z 305.003,A -85,B 0,C 180,E1 -380.981,E2 -380.981} C_VEL
LIN {X 0,Y 608.448,Z 305.008,A -85,B 0,C 180,E1 -383.124,E2 -383.124} C_VEL
LIN {X 0,Y 608.429,Z 305.006,A -85,B 0,C 180,E1 -385.719,E2 -385.719} C_VEL
LIN {X 0,Y 608.466,Z 305.008,A -85,B 0,C 180,E1 -388.624,E2 -388.624} C_VEL
LIN {X 0,Y 608.453,Z 305.002,A -85,B 0,C 180,E1 -391.317,E2 -391.317} C_VEL
LIN {X 0,Y 608.466,Z 305.008,A -85,B 0,C 180,E1 -393.739,E2 -393.739} C_VEL
LIN {X 0,Y 608.46,Z 305.003,A -85,B 0,C 180,E1 -396.091,E2 -396.091} C_VEL
LIN {X 0,Y 608.465,Z 305.003,A -85,B 0,C 180,E1 -398.588,E2 -398.588} C_VEL
LIN {X 0,Y 608.422,Z 305.007,A -85,B 0,C 180,E1 -401.342,E2 -401.342} C_VEL
LIN {X 0,Y 608.446,Z 305.011,A -85,B 0,C 180,E1 -404.266,E2 -404.266} C_VEL
LIN {X 0,Y 608.433,Z 305.005,A -85,B 0,C 180,E1 -407.042,E2 -407.042} C_VEL
LIN {X 0,Y 608.448,Z 305.009,A -85,B 0,C 180,E1 -409.699,E2 -409.699} C_VEL
LIN {X 0,Y 608.461,Z 305.001,A -85,B 0,C 180,E1 -412.256,E2 -412.256} C_VEL
LIN {X 0,Y 608.45,Z 305.008,A -85,B 0,C 180,E1 -415.094,E2 -415.094} C_VEL
LIN {X 0,Y 608.446,Z 305.164,A -85,B 0,C 180,E1 -415.45,E2 -415.45} C_VEL
LIN {X 0,Y 608.866,Z 308.721,A -85,B 0,C 180,E1 -415.958,E2 -415.958} C_VEL
LIN {X 0,Y 608.802,Z 329.264,A -85,B 0,C 180,E1 -418.677,E2 -418.677} C_VEL
LIN {X 0,Y 608.755,Z 349.881,A -85,B 0,C 180,E1 -421.331,E2 -421.331} C_VEL
LIN {X 0,Y 608.692,Z 373.053,A -85,B 0,C 180,E1 -424.236,E2 -424.236} C_VEL
LIN {X 0,Y 608.622,Z 396.319,A -85,B 0,C 180,E1 -427.083,E2 -427.083} C_VEL
LIN {X 0,Y 608.576,Z 420.624,A -85,B 0,C 180,E1 -429.996,E2 -429.996} C_VEL
LIN {X 0,Y 608.829,Z 424.6,A -85,B 0,C 180,E1 -430.071,E2 -430.071} C_VEL
LIN {X 0,Y 608.788,Z 446.032,A -85,B 0,C 180,E1 -430.377,E2 -430.377} C_VEL
LIN {X 0,Y 608.739,Z 462.483,A -85,B 0,C 180,E1 -430.748,E2 -430.748} C_VEL
LIN {X 0,Y 608.736,Z 478.554,A -85,B 0,C 180,E1 -431.252,E2 -431.252} C_VEL
LIN {X 0,Y 608.7,Z 493.116,A -85,B 0,C 180,E1 -431.838,E2 -431.838} C_VEL
LIN {X 0,Y 608.663,Z 508.91,A -85,B 0,C 180,E1 -432.618,E2 -432.618} C_VEL
LIN {X 0,Y 608.596,Z 523.594,A -85,B 0,C 180,E1 -433.496,E2 -433.496} C_VEL
LIN {X 0,Y 608.567,Z 536.716,A -85,B 0,C 180,E1 -434.427,E2 -434.427} C_VEL
LIN {X 0,Y 608.524,Z 549.029,A -85,B 0,C 180,E1 -435.454,E2 -435.454} C_VEL
LIN {X 0,Y 608.496,Z 559.653,A -85,B 0,C 180,E1 -436.476,E2 -436.476} C_VEL
LIN {X 0,Y 608.47,Z 570.345,A -85,B 0,C 180,E1 -437.664,E2 -437.664} C_VEL
LIN {X 0,Y 608.472,Z 580.873,A -85,B 0,C 180,E1 -439.042,E2 -439.042} C_VEL
LIN {X 0,Y 608.466,Z 589.294,A -85,B 0,C 180,E1 -440.361,E2 -440.361} C_VEL
LIN {X 0,Y 608.452,Z 596.494,A -85,B 0,C 180,E1 -441.7,E2 -441.7} C_VEL
LIN {X 0,Y 608.436,Z 602.476,A -85,B 0,C 180,E1 -443.036,E2 -443.036} C_VEL
LIN {X 0,Y 608.435,Z 608.251,A -85,B 0,C 180,E1 -444.7,E2 -444.7} C_VEL
LIN {X 0,Y 608.43,Z 611.636,A -85,B 0,C 180,E1 -446.028,E2 -446.028} C_VEL
LIN {X 0,Y 608.412,Z 614.088,A -85,B 0,C 180,E1 -447.353,E2 -447.353} C_VEL
LIN {X 0,Y 608.44,Z 615.478,A -85,B 0,C 180,E1 -448.678,E2 -448.678} C_VEL
LIN {X 0,Y 608.429,Z 616,A -85,B 0,C 180,E1 -450.002,E2 -450.002} C_VEL
LIN {X 0,Y 608.441,Z 615.476,A -85,B 0,C 180,E1 -451.325,E2 -451.325} C_VEL
LIN {X 0,Y 608.412,Z 614.083,A -85,B 0,C 180,E1 -452.65,E2 -452.65} C_VEL
LIN {X 0,Y 608.43,Z 611.629,A -85,B 0,C 180,E1 -453.976,E2 -453.976} C_VEL
LIN {X 0,Y 608.435,Z 608.24,A -85,B 0,C 180,E1 -455.304,E2 -455.304} C_VEL
LIN {X 0,Y 608.438,Z 602.463,A -85,B 0,C 180,E1 -456.968,E2 -456.968} C_VEL
LIN {X 0,Y 608.444,Z 594.85,A -85,B 0,C 180,E1 -458.638,E2 -458.638} C_VEL
LIN {X 0,Y 608.461,Z 586.236,A -85,B 0,C 180,E1 -460.147,E2 -460.147} C_VEL
LIN {X 0,Y 608.467,Z 576.957,A -85,B 0,C 180,E1 -461.494,E2 -461.494} C_VEL
LIN {X 0,Y 608.491,Z 567.409,A -85,B 0,C 180,E1 -462.678,E2 -462.678} C_VEL
LIN {X 0,Y 608.524,Z 555.952,A -85,B 0,C 180,E1 -463.897,E2 -463.897} C_VEL
LIN {X 0,Y 608.554,Z 544.126,A -85,B 0,C 180,E1 -464.977,E2 -464.977} C_VEL
LIN {X 0,Y 608.607,Z 529.692,A -85,B 0,C 180,E1 -466.091,E2 -466.091} C_VEL
LIN {X 0,Y 608.624,Z 514.994,A -85,B 0,C 180,E1 -467.04,E2 -467.04} C_VEL
LIN {X 0,Y 608.687,Z 500.485,A -85,B 0,C 180,E1 -467.818,E2 -467.818} C_VEL
LIN {X 0,Y 608.717,Z 485.242,A -85,B 0,C 180,E1 -468.493,E2 -468.493} C_VEL
LIN {X 0,Y 608.738,Z 469.193,A -85,B 0,C 180,E1 -469.058,E2 -469.058} C_VEL
LIN {X 0,Y 608.774,Z 453.467,A -85,B 0,C 180,E1 -469.473,E2 -469.473} C_VEL
LIN {X 0,Y 608.821,Z 437.841,A -85,B 0,C 180,E1 -469.757,E2 -469.757} C_VEL
LIN {X 0,Y 608.676,Z 421.303,A -85,B 0,C 180,E1 -469.975,E2 -469.975} C_VEL
LIN {X 0,Y 608.577,Z 420.595,A -85,B 0,C 180,E1 -470.007,E2 -470.007} C_VEL
LIN {X 0,Y 608.631,Z 397.627,A -85,B 0,C 180,E1 -472.758,E2 -472.758} C_VEL
LIN {X 0,Y 608.679,Z 374.503,A -85,B 0,C 180,E1 -475.585,E2 -475.585} C_VEL
LIN {X 0,Y 608.745,Z 353.164,A -85,B 0,C 180,E1 -478.253,E2 -478.253} C_VEL
LIN {X 0,Y 608.793,Z 332.416,A -85,B 0,C 180,E1 -480.913,E2 -480.913} C_VEL
LIN {X 0,Y 608.871,Z 311.668,A -85,B 0,C 180,E1 -483.646,E2 -483.646} C_VEL
LIN {X 0,Y 608.854,Z 307.222,A -85,B 0,C 180,E1 -484.245,E2 -484.245} C_VEL
LIN {X 0,Y 608.457,Z 305.008,A -85,B 0,C 180,E1 -484.581,E2 -484.581} C_VEL
LIN {X 0,Y 608.459,Z 305.005,A -85,B 0,C 180,E1 -487.157,E2 -487.157} C_VEL
LIN {X 0,Y 608.479,Z 305.003,A -85,B 0,C 180,E1 -489.44,E2 -489.44} C_VEL
LIN {X 0,Y 608.428,Z 305.009,A -85,B 0,C 180,E1 -492.331,E2 -492.331} C_VEL
LIN {X 0,Y 608.451,Z 305.009,A -85,B 0,C 180,E1 -494.797,E2 -494.797} C_VEL
LIN {X 0,Y 608.431,Z 305.01,A -85,B 0,C 180,E1 -497.039,E2 -497.039} C_VEL
LIN {X 0,Y 608.456,Z 305.006,A -85,B 0,C 180,E1 -499.697,E2 -499.697} C_VEL
LIN {X 0,Y 608.476,Z 305.007,A -85,B 0,C 180,E1 -502.842,E2 -502.842} C_VEL
LIN {X 0,Y 608.478,Z 305.046,A -85,B 0,C 180,E1 -505.423,E2 -505.423} C_VEL
LIN {X 0,Y 608.467,Z 310.714,A -85,B 0,C 180,E1 -507.478,E2 -507.478} C_VEL
LIN {X 0,Y 608.491,Z 316.873,A -85,B 0,C 180,E1 -510.026,E2 -510.026} C_VEL
LIN {X 0,Y 608.443,Z 322.331,A -85,B 0,C 180,E1 -512.482,E2 -512.482} C_VEL
LIN {X 0,Y 608.451,Z 329.173,A -85,B 0,C 180,E1 -515.429,E2 -515.429} C_VEL
LIN {X 0,Y 608.412,Z 336.016,A -85,B 0,C 180,E1 -518.307,E2 -518.307} C_VEL
LIN {X 0,Y 608.39,Z 341.149,A -85,B 0,C 180,E1 -520.428,E2 -520.428} C_VEL
LIN {X 0,Y 608.398,Z 347.992,A -85,B 0,C 180,E1 -523.215,E2 -523.215} C_VEL
LIN {X 0,Y 608.38,Z 354.981,A -85,B 0,C 180,E1 -526.018,E2 -526.018} C_VEL
LIN {X 0,Y 608.421,Z 360.718,A -85,B 0,C 180,E1 -528.296,E2 -528.296} C_VEL
LIN {X 0,Y 608.547,Z 374.365,A -85,B 0,C 180,E1 -528.593,E2 -528.593} C_VEL
LIN {X 0,Y 608.507,Z 387.644,A -85,B 0,C 180,E1 -529.028,E2 -529.028} C_VEL
LIN {X 0,Y 608.484,Z 398.74,A -85,B 0,C 180,E1 -529.519,E2 -529.519} C_VEL
LIN {X 0,Y 608.478,Z 410.516,A -85,B 0,C 180,E1 -530.191,E2 -530.191} C_VEL
LIN {X 0,Y 608.485,Z 421.028,A -85,B 0,C 180,E1 -530.946,E2 -530.946} C_VEL
LIN {X 0,Y 608.475,Z 429.637,A -85,B 0,C 180,E1 -531.699,E2 -531.699} C_VEL
LIN {X 0,Y 608.47,Z 437.566,A -85,B 0,C 180,E1 -532.534,E2 -532.534} C_VEL
LIN {X 0,Y 608.468,Z 445.073,A -85,B 0,C 180,E1 -533.498,E2 -533.498} C_VEL
LIN {X 0,Y 608.451,Z 450.611,A -85,B 0,C 180,E1 -534.366,E2 -534.366} C_VEL
LIN {X 0,Y 608.431,Z 455.753,A -85,B 0,C 180,E1 -535.362,E2 -535.362} C_VEL
LIN {X 0,Y 608.448,Z 459.742,A -85,B 0,C 180,E1 -536.358,E2 -536.358} C_VEL
LIN {X 0,Y 608.425,Z 462.691,A -85,B 0,C 180,E1 -537.352,E2 -537.352} C_VEL
LIN {X 0,Y 608.442,Z 464.127,A -85,B 0,C 180,E1 -538.014,E2 -538.014} C_VEL
LIN {X 0,Y 608.439,Z 465.752,A -85,B 0,C 180,E1 -539.338,E2 -539.338} C_VEL
LIN {X 0,Y 608.434,Z 465.995,A -85,B 0,C 180,E1 -540,E2 -540} C_VEL
LIN {X 0,Y 608.438,Z 465.815,A -85,B 0,C 180,E1 -540.662,E2 -540.662} C_VEL
LIN {X 0,Y 608.441,Z 464.276,A -85,B 0,C 180,E1 -541.986,E2 -541.986} C_VEL
LIN {X 0,Y 608.426,Z 462.918,A -85,B 0,C 180,E1 -542.649,E2 -542.649} C_VEL
LIN {X 0,Y 608.449,Z 460.041,A -85,B 0,C 180,E1 -543.643,E2 -543.643} C_VEL
LIN {X 0,Y 608.433,Z 456.142,A -85,B 0,C 180,E1 -544.638,E2 -544.638} C_VEL
LIN {X 0,Y 608.449,Z 451.111,A -85,B 0,C 180,E1 -545.635,E2 -545.635} C_VEL
LIN {X 0,Y 608.441,Z 444.793,A -85,B 0,C 180,E1 -546.633,E2 -546.633} C_VEL
LIN {X 0,Y 608.476,Z 436.876,A -85,B 0,C 180,E1 -547.633,E2 -547.633} C_VEL
LIN {X 0,Y 608.472,Z 427.033,A -85,B 0,C 180,E1 -548.636,E2 -548.636} C_VEL
LIN {X 0,Y 608.477,Z 424.939,A -85,B 0,C 180,E1 -548.819,E2 -548.819} C_VEL
LIN {X 0,Y 607.81,Z 420.606,A -85,B 0,C 180,E1 -549.189,E2 -549.189} C_VEL
LIN {X 0,Y 604.965,Z 413.359,A -85,B 0,C 180,E1 -549.769,E2 -549.769} C_VEL
LIN {X 0,Y 602.134,Z 405.719,A -85,B 0,C 180,E1 -550.301,E2 -550.301} C_VEL
LIN {X 0,Y 601.492,Z 400.657,A -85,B 0,C 180,E1 -550.594,E2 -550.594} C_VEL
LIN {X 0,Y 601.544,Z 388.845,A -85,B 0,C 180,E1 -551.145,E2 -551.145} C_VEL
LIN {X 0,Y 601.594,Z 376.049,A -85,B 0,C 180,E1 -551.583,E2 -551.583} C_VEL
LIN {X 0,Y 601.585,Z 362.623,A -85,B 0,C 180,E1 -551.893,E2 -551.893} C_VEL
LIN {X 0,Y 601.329,Z 360.675,A -85,B 0,C 180,E1 -551.952,E2 -551.952} C_VEL
LIN {X 0,Y 601.349,Z 353.348,A -85,B 0,C 180,E1 -554.899,E2 -554.899} C_VEL
LIN {X 0,Y 601.326,Z 346.501,A -85,B 0,C 180,E1 -557.691,E2 -557.691} C_VEL
LIN {X 0,Y 601.348,Z 339.654,A -85,B 0,C 180,E1 -560.525,E2 -560.525} C_VEL
LIN {X 0,Y 601.365,Z 332.806,A -85,B 0,C 180,E1 -563.413,E2 -563.413} C_VEL
LIN {X 0,Y 601.367,Z 327.126,A -85,B 0,C 180,E1 -565.857,E2 -565.857} C_VEL
LIN {X 0,Y 601.432,Z 320.502,A -85,B 0,C 180,E1 -568.787,E2 -568.787} C_VEL
LIN {X 0,Y 601.449,Z 314.575,A -85,B 0,C 180,E1 -571.458,E2 -571.458} C_VEL
LIN {X 0,Y 601.435,Z 308.684,A -85,B 0,C 180,E1 -574.118,E2 -574.118} C_VEL
LIN {X 0,Y 601.423,Z 305.884,A -85,B 0,C 180,E1 -575.405,E2 -575.405} C_VEL
LIN {X 0,Y 601.417,Z 305.883,A -85,B 0,C 180,E1 -578.269,E2 -578.269} C_VEL
LIN {X 0,Y 601.417,Z 305.883,A -85,B 0,C 180,E1 -580.875,E2 -580.875} C_VEL
LIN {X 0,Y 601.413,Z 305.884,A -85,B 0,C 180,E1 -583.588,E2 -583.588} C_VEL
LIN {X 0,Y 601.413,Z 305.887,A -85,B 0,C 180,E1 -586.429,E2 -586.429} C_VEL
LIN {X 0,Y 601.419,Z 305.886,A -85,B 0,C 180,E1 -589.125,E2 -589.125} C_VEL
LIN {X 0,Y 601.416,Z 305.886,A -85,B 0,C 180,E1 -591.731,E2 -591.731} C_VEL
LIN {X 0,Y 601.394,Z 305.889,A -85,B 0,C 180,E1 -594.245,E2 -594.245} C_VEL
LIN {X 0,Y 601.418,Z 305.902,A -85,B 0,C 180,E1 -595.067,E2 -595.067} C_VEL
LIN {X 0,Y 601.433,Z 311.831,A -85,B 0,C 180,E1 -597.483,E2 -597.483} C_VEL
LIN {X 0,Y 601.41,Z 317.261,A -85,B 0,C 180,E1 -599.855,E2 -599.855} C_VEL
LIN {X 0,Y 601.369,Z 324.04,A -85,B 0,C 180,E1 -602.884,E2 -602.884} C_VEL
LIN {X 0,Y 601.366,Z 329.172,A -85,B 0,C 180,E1 -605.119,E2 -605.119} C_VEL
LIN {X 0,Y 601.372,Z 334.519,A -85,B 0,C 180,E1 -607.405,E2 -607.405} C_VEL
LIN {X 0,Y 601.364,Z 341.147,A -85,B 0,C 180,E1 -610.188,E2 -610.188} C_VEL
LIN {X 0,Y 601.356,Z 347.99,A -85,B 0,C 180,E1 -613.011,E2 -613.011} C_VEL
LIN {X 0,Y 601.354,Z 355.19,A -85,B 0,C 180,E1 -615.935,E2 -615.935} C_VEL
LIN {X 0,Y 601.352,Z 360.715,A -85,B 0,C 180,E1 -618.154,E2 -618.154} C_VEL
LIN {X 0,Y 601.592,Z 368.271,A -85,B 0,C 180,E1 -618.309,E2 -618.309} C_VEL
LIN {X 0,Y 601.532,Z 381.134,A -85,B 0,C 180,E1 -618.664,E2 -618.664} C_VEL
LIN {X 0,Y 601.487,Z 393.134,A -85,B 0,C 180,E1 -619.129,E2 -619.129} C_VEL
LIN {X 0,Y 601.487,Z 404.991,A -85,B 0,C 180,E1 -619.734,E2 -619.734} C_VEL
LIN {X 0,Y 601.462,Z 416.62,A -85,B 0,C 180,E1 -620.499,E2 -620.499} C_VEL
LIN {X 0,Y 601.437,Z 426.007,A -85,B 0,C 180,E1 -621.261,E2 -621.261} C_VEL
LIN {X 0,Y 601.401,Z 434.561,A -85,B 0,C 180,E1 -622.106,E2 -622.106} C_VEL
LIN {X 0,Y 601.384,Z 442.896,A -85,B 0,C 180,E1 -623.119,E2 -623.119} C_VEL
LIN {X 0,Y 601.373,Z 449.6,A -85,B 0,C 180,E1 -624.129,E2 -624.129} C_VEL
LIN {X 0,Y 601.335,Z 455.743,A -85,B 0,C 180,E1 -625.306,E2 -625.306} C_VEL
LIN {X 0,Y 601.367,Z 459.735,A -85,B 0,C 180,E1 -626.313,E2 -626.313} C_VEL
LIN {X 0,Y 601.324,Z 462.69,A -85,B 0,C 180,E1 -627.319,E2 -627.319} C_VEL
LIN {X 0,Y 601.343,Z 464.126,A -85,B 0,C 180,E1 -627.989,E2 -627.989} C_VEL
LIN {X 0,Y 601.339,Z 465.752,A -85,B 0,C 180,E1 -629.329,E2 -629.329} C_VEL
LIN {X 0,Y 601.336,Z 465.995,A -85,B 0,C 180,E1 -629.998,E2 -629.998} C_VEL
LIN {X 0,Y 601.339,Z 465.817,A -85,B 0,C 180,E1 -630.668,E2 -630.668} C_VEL
LIN {X 0,Y 601.343,Z 464.279,A -85,B 0,C 180,E1 -632.008,E2 -632.008} C_VEL
LIN {X 0,Y 601.326,Z 462.912,A -85,B 0,C 180,E1 -632.678,E2 -632.678} C_VEL
LIN {X 0,Y 601.368,Z 460.038,A -85,B 0,C 180,E1 -633.684,E2 -633.684} C_VEL
LIN {X 0,Y 601.336,Z 456.14,A -85,B 0,C 180,E1 -634.691,E2 -634.691} C_VEL
LIN {X 0,Y 601.373,Z 451.114,A -85,B 0,C 180,E1 -635.699,E2 -635.699} C_VEL
LIN {X 0,Y 601.381,Z 444.803,A -85,B 0,C 180,E1 -636.709,E2 -636.709} C_VEL
LIN {X 0,Y 601.395,Z 436.89,A -85,B 0,C 180,E1 -637.722,E2 -637.722} C_VEL
LIN {X 0,Y 601.422,Z 428.826,A -85,B 0,C 180,E1 -638.567,E2 -638.567} C_VEL
LIN {X 0,Y 601.453,Z 418.988,A -85,B 0,C 180,E1 -639.414,E2 -639.414} C_VEL
LIN {X 0,Y 601.476,Z 407.952,A -85,B 0,C 180,E1 -640.177,E2 -640.177} C_VEL
LIN {X 0,Y 601.477,Z 395.252,A -85,B 0,C 180,E1 -640.865,E2 -640.865} C_VEL
LIN {X 0,Y 601.521,Z 382.732,A -85,B 0,C 180,E1 -641.373,E2 -641.373} C_VEL
LIN {X 0,Y 601.592,Z 370.437,A -85,B 0,C 180,E1 -641.731,E2 -641.731} C_VEL
LIN {X 0,Y 601.353,Z 360.828,A -85,B 0,C 180,E1 -641.928,E2 -641.928} C_VEL
LIN {X 0,Y 601.353,Z 353.353,A -85,B 0,C 180,E1 -644.897,E2 -644.897} C_VEL
LIN {X 0,Y 601.362,Z 346.507,A -85,B 0,C 180,E1 -647.687,E2 -647.687} C_VEL
LIN {X 0,Y 601.368,Z 339.66,A -85,B 0,C 180,E1 -650.522,E2 -650.522} C_VEL
LIN {X 0,Y 601.378,Z 332.812,A -85,B 0,C 180,E1 -653.41,E2 -653.41} C_VEL
LIN {X 0,Y 601.397,Z 327.108,A -85,B 0,C 180,E1 -655.863,E2 -655.863} C_VEL
LIN {X 0,Y 601.377,Z 320.519,A -85,B 0,C 180,E1 -658.778,E2 -658.778} C_VEL
LIN {X 0,Y 601.438,Z 314.489,A -85,B 0,C 180,E1 -661.457,E2 -661.457} C_VEL
LIN {X 0,Y 601.428,Z 308.229,A -85,B 0,C 180,E1 -664.116,E2 -664.116} C_VEL
LIN {X 0,Y 601.412,Z 305.883,A -85,B 0,C 180,E1 -665.114,E2 -665.114} C_VEL
LIN {X 0,Y 601.426,Z 305.878,A -85,B 0,C 180,E1 -667.417,E2 -667.417} C_VEL
LIN {X 0,Y 601.398,Z 305.889,A -85,B 0,C 180,E1 -669.993,E2 -669.993} C_VEL
LIN {X 0,Y 601.357,Z 305.886,A -85,B 0,C 180,E1 -672.672,E2 -672.672} C_VEL
LIN {X 0,Y 601.41,Z 305.883,A -85,B 0,C 180,E1 -675.48,E2 -675.48} C_VEL
LIN {X 0,Y 601.415,Z 305.883,A -85,B 0,C 180,E1 -678.404,E2 -678.404} C_VEL
LIN {X 0,Y 601.424,Z 305.88,A -85,B 0,C 180,E1 -680.874,E2 -680.874} C_VEL
LIN {X 0,Y 601.428,Z 305.883,A -85,B 0,C 180,E1 -683.732,E2 -683.732} C_VEL
LIN {X 0,Y 601.391,Z 305.882,A -85,B 0,C 180,E1 -686.684,E2 -686.684} C_VEL
LIN {X 0,Y 601.394,Z 305.888,A -85,B 0,C 180,E1 -689.056,E2 -689.056} C_VEL
LIN {X 0,Y 601.425,Z 305.88,A -85,B 0,C 180,E1 -691.373,E2 -691.373} C_VEL
LIN {X 0,Y 601.397,Z 305.881,A -85,B 0,C 180,E1 -693.636,E2 -693.636} C_VEL
LIN {X 0,Y 601.414,Z 305.881,A -85,B 0,C 180,E1 -696.589,E2 -696.589} C_VEL
LIN {X 0,Y 601.427,Z 305.883,A -85,B 0,C 180,E1 -699.478,E2 -699.478} C_VEL
LIN {X 0,Y 601.359,Z 305.886,A -85,B 0,C 180,E1 -702.31,E2 -702.31} C_VEL
LIN {X 0,Y 601.388,Z 305.884,A -85,B 0,C 180,E1 -704.408,E2 -704.408} C_VEL
LIN {X 0,Y 601.412,Z 305.88,A -85,B 0,C 180,E1 -707.171,E2 -707.171} C_VEL
LIN {X 0,Y 601.434,Z 305.881,A -85,B 0,C 180,E1 -709.905,E2 -709.905} C_VEL
LIN {X 0,Y 601.435,Z 305.877,A -85,B 0,C 180,E1 -712.615,E2 -712.615} C_VEL
LIN {X 0,Y 601.424,Z 305.885,A -85,B 0,C 180,E1 -715.308,E2 -715.308} C_VEL
LIN {X 0,Y 601.374,Z 305.884,A -85,B 0,C 180,E1 -717.991,E2 -717.991} C_VEL
LIN {X 0,Y 601.448,Z 305.882,A -85,B 0,C 180,E1 -720.669,E2 -720.669} C_VEL
LIN {X 0,Y 601.421,Z 305.878,A -85,B 0,C 180,E1 -723.349,E2 -723.349} C_VEL
LIN {X 0,Y 601.435,Z 305.882,A -85,B 0,C 180,E1 -726.037,E2 -726.037} C_VEL
LIN {X 0,Y 601.421,Z 305.879,A -85,B 0,C 180,E1 -728.738,E2 -728.738} C_VEL
LIN {X 0,Y 601.408,Z 305.883,A -85,B 0,C 180,E1 -731.458,E2 -731.458} C_VEL
LIN {X 0,Y 601.385,Z 305.885,A -85,B 0,C 180,E1 -734.206,E2 -734.206} C_VEL
LIN {X 0,Y 601.418,Z 305.879,A -85,B 0,C 180,E1 -736.986,E2 -736.986} C_VEL
LIN {X 0,Y 601.397,Z 305.89,A -85,B 0,C 180,E1 -739.809,E2 -739.809} C_VEL
LIN {X 0,Y 601.434,Z 305.877,A -85,B 0,C 180,E1 -742.682,E2 -742.682} C_VEL
LIN {X 0,Y 601.387,Z 305.888,A -85,B 0,C 180,E1 -744.879,E2 -744.879} C_VEL
LIN {X 0,Y 601.375,Z 305.884,A -85,B 0,C 180,E1 -747.869,E2 -747.869} C_VEL
LIN {X 0,Y 601.404,Z 305.886,A -85,B 0,C 180,E1 -750.165,E2 -750.165} C_VEL
LIN {X 0,Y 601.417,Z 305.879,A -85,B 0,C 180,E1 -752.72,E2 -752.72} C_VEL
LIN {X 0,Y 601.41,Z 305.882,A -85,B 0,C 180,E1 -755.118,E2 -755.118} C_VEL
LIN {X 0,Y 601.419,Z 305.885,A -85,B 0,C 180,E1 -757.42,E2 -757.42} C_VEL
LIN {X 0,Y 601.392,Z 305.882,A -85,B 0,C 180,E1 -759.996,E2 -759.996} C_VEL
LIN {X 0,Y 601.386,Z 305.889,A -85,B 0,C 180,E1 -762.672,E2 -762.672} C_VEL
LIN {X 0,Y 601.407,Z 305.882,A -85,B 0,C 180,E1 -765.484,E2 -765.484} C_VEL
LIN {X 0,Y 601.42,Z 305.88,A -85,B 0,C 180,E1 -768.407,E2 -768.407} C_VEL
LIN {X 0,Y 601.428,Z 305.881,A -85,B 0,C 180,E1 -770.878,E2 -770.878} C_VEL
LIN {X 0,Y 601.418,Z 305.881,A -85,B 0,C 180,E1 -773.737,E2 -773.737} C_VEL
LIN {X 0,Y 601.414,Z 305.954,A -85,B 0,C 180,E1 -775.096,E2 -775.096} C_VEL
LIN {X 0,Y 602.267,Z 310.215,A -85,B 0,C 180,E1 -775.737,E2 -775.737} C_VEL
LIN {X 0,Y 602.14,Z 330.342,A -85,B 0,C 180,E1 -778.433,E2 -778.433} C_VEL
LIN {X 0,Y 601.999,Z 351.944,A -85,B 0,C 180,E1 -781.245,E2 -781.245} C_VEL
LIN {X 0,Y 601.881,Z 373.992,A -85,B 0,C 180,E1 -784.04,E2 -784.04} C_VEL
LIN {X 0,Y 601.793,Z 394.689,A -85,B 0,C 180,E1 -786.607,E2 -786.607} C_VEL
LIN {X 0,Y 601.67,Z 418.401,A -85,B 0,C 180,E1 -789.489,E2 -789.489} C_VEL
LIN {X 0,Y 601.655,Z 420.716,A -85,B 0,C 180,E1 -789.767,E2 -789.767} C_VEL
LIN {X 0,Y 602.161,Z 424.6,A -85,B 0,C 180,E1 -789.841,E2 -789.841} C_VEL
LIN {X 0,Y 602.122,Z 446.032,A -85,B 0,C 180,E1 -790.151,E2 -790.151} C_VEL
LIN {X 0,Y 602.043,Z 461.721,A -85,B 0,C 180,E1 -790.503,E2 -790.503} C_VEL
LIN {X 0,Y 602.007,Z 478.032,A -85,B 0,C 180,E1 -791.016,E2 -791.016} C_VEL
LIN {X 0,Y 601.893,Z 493.118,A -85,B 0,C 180,E1 -791.625,E2 -791.625} C_VEL
LIN {X 0,Y 601.802,Z 508.911,A -85,B 0,C 180,E1 -792.414,E2 -792.414} C_VEL
LIN {X 0,Y 601.721,Z 523.327,A -85,B 0,C 180,E1 -793.284,E2 -793.284} C_VEL
LIN {X 0,Y 601.66,Z 536.717,A -85,B 0,C 180,E1 -794.244,E2 -794.244} C_VEL
LIN {X 0,Y 601.582,Z 549.029,A -85,B 0,C 180,E1 -795.282,E2 -795.282} C_VEL
LIN {X 0,Y 601.489,Z 561.281,A -85,B 0,C 180,E1 -796.488,E2 -796.488} C_VEL
LIN {X 0,Y 601.451,Z 571.707,A -85,B 0,C 180,E1 -797.689,E2 -797.689} C_VEL
LIN {X 0,Y 601.424,Z 581.372,A -85,B 0,C 180,E1 -798.987,E2 -798.987} C_VEL
LIN {X 0,Y 601.393,Z 589.295,A -85,B 0,C 180,E1 -800.246,E2 -800.246} C_VEL
LIN {X 0,Y 601.364,Z 596.495,A -85,B 0,C 180,E1 -801.602,E2 -801.602} C_VEL
LIN {X 0,Y 601.364,Z 602.475,A -85,B 0,C 180,E1 -802.953,E2 -802.953} C_VEL
LIN {X 0,Y 601.346,Z 608.251,A -85,B 0,C 180,E1 -804.637,E2 -804.637} C_VEL
LIN {X 0,Y 601.339,Z 611.636,A -85,B 0,C 180,E1 -805.981,E2 -805.981} C_VEL
LIN {X 0,Y 601.311,Z 614.089,A -85,B 0,C 180,E1 -807.322,E2 -807.322} C_VEL
LIN {X 0,Y 601.34,Z 615.478,A -85,B 0,C 180,E1 -808.662,E2 -808.662} C_VEL
LIN {X 0,Y 601.33,Z 616,A -85,B 0,C 180,E1 -810.002,E2 -810.002} C_VEL
LIN {X 0,Y 601.341,Z 615.476,A -85,B 0,C 180,E1 -811.341,E2 -811.341} C_VEL
LIN {X 0,Y 601.311,Z 614.083,A -85,B 0,C 180,E1 -812.681,E2 -812.681} C_VEL
LIN {X 0,Y 601.339,Z 611.629,A -85,B 0,C 180,E1 -814.023,E2 -814.023} C_VEL
LIN {X 0,Y 601.346,Z 608.241,A -85,B 0,C 180,E1 -815.366,E2 -815.366} C_VEL
LIN {X 0,Y 601.363,Z 602.463,A -85,B 0,C 180,E1 -817.05,E2 -817.05} C_VEL
LIN {X 0,Y 601.377,Z 594.85,A -85,B 0,C 180,E1 -818.74,E2 -818.74} C_VEL
LIN {X 0,Y 601.41,Z 586.237,A -85,B 0,C 180,E1 -820.267,E2 -820.267} C_VEL
LIN {X 0,Y 601.431,Z 576.958,A -85,B 0,C 180,E1 -821.63,E2 -821.63} C_VEL
LIN {X 0,Y 601.48,Z 567.41,A -85,B 0,C 180,E1 -822.828,E2 -822.828} C_VEL
LIN {X 0,Y 601.547,Z 556.605,A -85,B 0,C 180,E1 -823.998,E2 -823.998} C_VEL
LIN {X 0,Y 601.607,Z 544.127,A -85,B 0,C 180,E1 -825.154,E2 -825.154} C_VEL
LIN {X 0,Y 601.718,Z 529.692,A -85,B 0,C 180,E1 -826.28,E2 -826.28} C_VEL
LIN {X 0,Y 601.778,Z 514.996,A -85,B 0,C 180,E1 -827.24,E2 -827.24} C_VEL
LIN {X 0,Y 601.861,Z 500.487,A -85,B 0,C 180,E1 -828.027,E2 -828.027} C_VEL
LIN {X 0,Y 601.954,Z 485.019,A -85,B 0,C 180,E1 -828.717,E2 -828.717} C_VEL
LIN {X 0,Y 602.025,Z 469.195,A -85,B 0,C 180,E1 -829.279,E2 -829.279} C_VEL
LIN {X 0,Y 602.096,Z 452.552,A -85,B 0,C 180,E1 -829.72,E2 -829.72} C_VEL
LIN {X 0,Y 602.14,Z 436.335,A -85,B 0,C 180,E1 -830.008,E2 -830.008} C_VEL
LIN {X 0,Y 602.03,Z 422.533,A -85,B 0,C 180,E1 -830.19,E2 -830.19} C_VEL
LIN {X 0,Y 601.652,Z 420.595,A -85,B 0,C 180,E1 -830.247,E2 -830.247} C_VEL
LIN {X 0,Y 601.77,Z 399.255,A -85,B 0,C 180,E1 -832.833,E2 -832.833} C_VEL
LIN {X 0,Y 601.858,Z 376.876,A -85,B 0,C 180,E1 -835.599,E2 -835.599} C_VEL
LIN {X 0,Y 601.973,Z 356.128,A -85,B 0,C 180,E1 -838.22,E2 -838.22} C_VEL
LIN {X 0,Y 602.115,Z 335.38,A -85,B 0,C 180,E1 -840.903,E2 -840.903} C_VEL
LIN {X 0,Y 602.224,Z 314.632,A -85,B 0,C 180,E1 -843.666,E2 -843.666} C_VEL
LIN {X 0,Y 602.101,Z 308.704,A -85,B 0,C 180,E1 -844.481,E2 -844.481} C_VEL
LIN {X 0,Y 601.441,Z 305.884,A -85,B 0,C 180,E1 -844.931,E2 -844.931} C_VEL
LIN {X 0,Y 601.431,Z 305.883,A -85,B 0,C 180,E1 -847.42,E2 -847.42} C_VEL
LIN {X 0,Y 601.415,Z 305.883,A -85,B 0,C 180,E1 -849.996,E2 -849.996} C_VEL
LIN {X 0,Y 601.382,Z 305.887,A -85,B 0,C 180,E1 -852.674,E2 -852.674} C_VEL
LIN {X 0,Y 601.431,Z 305.881,A -85,B 0,C 180,E1 -855.483,E2 -855.483} C_VEL
LIN {X 0,Y 601.419,Z 305.883,A -85,B 0,C 180,E1 -858.408,E2 -858.408} C_VEL
LIN {X 0,Y 601.397,Z 305.885,A -85,B 0,C 180,E1 -860.873,E2 -860.873} C_VEL
LIN {X 0,Y 601.41,Z 305.884,A -85,B 0,C 180,E1 -863.418,E2 -863.418} C_VEL
LIN {X 0,Y 601.432,Z 306.042,A -85,B 0,C 180,E1 -865.477,E2 -865.477} C_VEL
LIN {X 0,Y 601.423,Z 312.604,A -85,B 0,C 180,E1 -867.88,E2 -867.88} C_VEL
LIN {X 0,Y 601.428,Z 319.168,A -85,B 0,C 180,E1 -870.608,E2 -870.608} C_VEL
LIN {X 0,Y 601.389,Z 324.043,A -85,B 0,C 180,E1 -872.886,E2 -872.886} C_VEL
LIN {X 0,Y 601.382,Z 330.568,A -85,B 0,C 180,E1 -875.72,E2 -875.72} C_VEL
LIN {X 0,Y 601.341,Z 336.018,A -85,B 0,C 180,E1 -878.038,E2 -878.038} C_VEL
LIN {X 0,Y 601.33,Z 341.15,A -85,B 0,C 180,E1 -880.188,E2 -880.188} C_VEL
LIN {X 0,Y 601.324,Z 346.283,A -85,B 0,C 180,E1 -882.31,E2 -882.31} C_VEL
LIN {X 0,Y 601.344,Z 353.127,A -85,B 0,C 180,E1 -885.101,E2 -885.101} C_VEL
LIN {X 0,Y 601.326,Z 360.719,A -85,B 0,C 180,E1 -888.155,E2 -888.155} C_VEL
LIN {X 0,Y 601.615,Z 370.182,A -85,B 0,C 180,E1 -888.353,E2 -888.353} C_VEL
LIN {X 0,Y 601.571,Z 383.391,A -85,B 0,C 180,E1 -888.739,E2 -888.739} C_VEL
LIN {X 0,Y 601.504,Z 395.254,A -85,B 0,C 180,E1 -889.226,E2 -889.226} C_VEL
LIN {X 0,Y 601.47,Z 406.426,A -85,B 0,C 180,E1 -889.821,E2 -889.821} C_VEL
LIN {X 0,Y 601.455,Z 417.802,A -85,B 0,C 180,E1 -890.585,E2 -890.585} C_VEL
LIN {X 0,Y 601.424,Z 427.867,A -85,B 0,C 180,E1 -891.432,E2 -891.432} C_VEL
LIN {X 0,Y 601.418,Z 437.571,A -85,B 0,C 180,E1 -892.446,E2 -892.446} C_VEL
LIN {X 0,Y 601.377,Z 444.892,A -85,B 0,C 180,E1 -893.393,E2 -893.393} C_VEL
LIN {X 0,Y 601.372,Z 450.614,A -85,B 0,C 180,E1 -894.299,E2 -894.299} C_VEL
LIN {X 0,Y 601.336,Z 455.755,A -85,B 0,C 180,E1 -895.308,E2 -895.308} C_VEL
LIN {X 0,Y 601.367,Z 459.744,A -85,B 0,C 180,E1 -896.315,E2 -896.315} C_VEL
LIN {X 0,Y 601.324,Z 462.693,A -85,B 0,C 180,E1 -897.321,E2 -897.321} C_VEL
LIN {X 0,Y 601.341,Z 464.128,A -85,B 0,C 180,E1 -897.991,E2 -897.991} C_VEL
LIN {X 0,Y 601.339,Z 465.753,A -85,B 0,C 180,E1 -899.331,E2 -899.331} C_VEL
LIN {X 0,Y 601.335,Z 465.996,A -85,B 0,C 180,E1 -900,E2 -900} C_VEL
LIN {X 0,Y 601.339,Z 465.815,A -85,B 0,C 180,E1 -900.67,E2 -900.67} C_VEL
LIN {X 0,Y 601.34,Z 464.275,A -85,B 0,C 180,E1 -902.01,E2 -902.01} C_VEL
LIN {X 0,Y 601.326,Z 462.917,A -85,B 0,C 180,E1 -902.68,E2 -902.68} C_VEL
LIN {X 0,Y 601.368,Z 460.039,A -85,B 0,C 180,E1 -903.686,E2 -903.686} C_VEL
LIN {X 0,Y 601.337,Z 456.139,A -85,B 0,C 180,E1 -904.693,E2 -904.693} C_VEL
LIN {X 0,Y 601.373,Z 451.109,A -85,B 0,C 180,E1 -905.701,E2 -905.701} C_VEL
LIN {X 0,Y 601.383,Z 444.789,A -85,B 0,C 180,E1 -906.711,E2 -906.711} C_VEL
LIN {X 0,Y 601.396,Z 436.872,A -85,B 0,C 180,E1 -907.724,E2 -907.724} C_VEL
LIN {X 0,Y 601.437,Z 427.027,A -85,B 0,C 180,E1 -908.738,E2 -908.738} C_VEL
LIN {X 0,Y 601.446,Z 416.704,A -85,B 0,C 180,E1 -909.585,E2 -909.585} C_VEL
LIN {X 0,Y 601.468,Z 405.085,A -85,B 0,C 180,E1 -910.35,E2 -910.35} C_VEL
LIN {X 0,Y 601.492,Z 400.657,A -85,B 0,C 180,E1 -910.594,E2 -910.594} C_VEL
LIN {X 0,Y 600.87,Z 395.529,A -85,B 0,C 180,E1 -910.869,E2 -910.869} C_VEL
LIN {X 0,Y 598.123,Z 387.069,A -85,B 0,C 180,E1 -911.288,E2 -911.288} C_VEL
LIN {X 0,Y 595.336,Z 378.314,A -85,B 0,C 180,E1 -911.643,E2 -911.643} C_VEL
LIN {X 0,Y 594.649,Z 372.728,A -85,B 0,C 180,E1 -911.814,E2 -911.814} C_VEL
LIN {X 0,Y 594.417,Z 362.022,A -85,B 0,C 180,E1 -912.05,E2 -912.05} C_VEL
LIN {X 0,Y 594.255,Z 360.728,A -85,B 0,C 180,E1 -912.075,E2 -912.075} C_VEL
LIN {X 0,Y 594.262,Z 353.346,A -85,B 0,C 180,E1 -915.081,E2 -915.081} C_VEL
LIN {X 0,Y 594.235,Z 346.499,A -85,B 0,C 180,E1 -917.909,E2 -917.909} C_VEL
LIN {X 0,Y 594.306,Z 339.652,A -85,B 0,C 180,E1 -920.779,E2 -920.779} C_VEL
LIN {X 0,Y 594.29,Z 332.805,A -85,B 0,C 180,E1 -923.709,E2 -923.709} C_VEL
LIN {X 0,Y 594.3,Z 327.54,A -85,B 0,C 180,E1 -926.005,E2 -926.005} C_VEL
LIN {X 0,Y 594.344,Z 322.628,A -85,B 0,C 180,E1 -928.229,E2 -928.229} C_VEL
LIN {X 0,Y 594.39,Z 317.469,A -85,B 0,C 180,E1 -930.559,E2 -930.559} C_VEL
LIN {X 0,Y 594.389,Z 312.213,A -85,B 0,C 180,E1 -932.95,E2 -932.95} C_VEL
LIN {X 0,Y 594.388,Z 306.76,A -85,B 0,C 180,E1 -935.511,E2 -935.511} C_VEL
LIN {X 0,Y 594.386,Z 306.76,A -85,B 0,C 180,E1 -937.941,E2 -937.941} C_VEL
LIN {X 0,Y 594.381,Z 306.759,A -85,B 0,C 180,E1 -940.821,E2 -940.821} C_VEL
LIN {X 0,Y 594.357,Z 306.762,A -85,B 0,C 180,E1 -943.301,E2 -943.301} C_VEL
LIN {X 0,Y 594.35,Z 306.764,A -85,B 0,C 180,E1 -946.163,E2 -946.163} C_VEL
LIN {X 0,Y 594.389,Z 306.758,A -85,B 0,C 180,E1 -948.536,E2 -948.536} C_VEL
LIN {X 0,Y 594.376,Z 306.761,A -85,B 0,C 180,E1 -951.297,E2 -951.297} C_VEL
LIN {X 0,Y 594.355,Z 306.764,A -85,B 0,C 180,E1 -953.755,E2 -953.755} C_VEL
LIN {X 0,Y 594.398,Z 306.81,A -85,B 0,C 180,E1 -955.008,E2 -955.008} C_VEL
LIN {X 0,Y 594.431,Z 311.927,A -85,B 0,C 180,E1 -957.081,E2 -957.081} C_VEL
LIN {X 0,Y 594.375,Z 317.805,A -85,B 0,C 180,E1 -959.674,E2 -959.674} C_VEL
LIN {X 0,Y 594.34,Z 324.099,A -85,B 0,C 180,E1 -962.536,E2 -962.536} C_VEL
LIN {X 0,Y 594.321,Z 329.173,A -85,B 0,C 180,E1 -964.803,E2 -964.803} C_VEL
LIN {X 0,Y 594.31,Z 336.016,A -85,B 0,C 180,E1 -967.763,E2 -967.763} C_VEL
LIN {X 0,Y 594.285,Z 342.859,A -85,B 0,C 180,E1 -970.662,E2 -970.662} C_VEL
LIN {X 0,Y 594.288,Z 349.702,A -85,B 0,C 180,E1 -973.51,E2 -973.51} C_VEL
LIN {X 0,Y 594.261,Z 356.546,A -85,B 0,C 180,E1 -976.317,E2 -976.317} C_VEL
LIN {X 0,Y 594.269,Z 360.716,A -85,B 0,C 180,E1 -978.011,E2 -978.011} C_VEL
LIN {X 0,Y 594.688,Z 365.221,A -85,B 0,C 180,E1 -978.106,E2 -978.106} C_VEL
LIN {X 0,Y 594.593,Z 378.766,A -85,B 0,C 180,E1 -978.45,E2 -978.45} C_VEL
LIN {X 0,Y 594.531,Z 391.279,A -85,B 0,C 180,E1 -978.919,E2 -978.919} C_VEL
LIN {X 0,Y 594.487,Z 401.905,A -85,B 0,C 180,E1 -979.44,E2 -979.44} C_VEL
LIN {X 0,Y 594.46,Z 413.051,A -85,B 0,C 180,E1 -980.128,E2 -980.128} C_VEL
LIN {X 0,Y 594.412,Z 424.076,A -85,B 0,C 180,E1 -980.985,E2 -980.985} C_VEL
LIN {X 0,Y 594.367,Z 432.973,A -85,B 0,C 180,E1 -981.841,E2 -981.841} C_VEL
LIN {X 0,Y 594.306,Z 441.638,A -85,B 0,C 180,E1 -982.866,E2 -982.866} C_VEL
LIN {X 0,Y 594.29,Z 448.595,A -85,B 0,C 180,E1 -983.889,E2 -983.889} C_VEL
LIN {X 0,Y 594.254,Z 454.15,A -85,B 0,C 180,E1 -984.91,E2 -984.91} C_VEL
LIN {X 0,Y 594.263,Z 458.512,A -85,B 0,C 180,E1 -985.929,E2 -985.929} C_VEL
LIN {X 0,Y 594.267,Z 460.802,A -85,B 0,C 180,E1 -986.608,E2 -986.608} C_VEL
LIN {X 0,Y 594.225,Z 462.69,A -85,B 0,C 180,E1 -987.287,E2 -987.287} C_VEL
LIN {X 0,Y 594.242,Z 464.129,A -85,B 0,C 180,E1 -987.965,E2 -987.965} C_VEL
LIN {X 0,Y 594.24,Z 465.753,A -85,B 0,C 180,E1 -989.321,E2 -989.321} C_VEL
LIN {X 0,Y 594.236,Z 465.995,A -85,B 0,C 180,E1 -989.998,E2 -989.998} C_VEL
LIN {X 0,Y 594.239,Z 465.815,A -85,B 0,C 180,E1 -990.676,E2 -990.676} C_VEL
LIN {X 0,Y 594.242,Z 464.28,A -85,B 0,C 180,E1 -992.032,E2 -992.032} C_VEL
LIN {X 0,Y 594.226,Z 462.903,A -85,B 0,C 180,E1 -992.71,E2 -992.71} C_VEL
LIN {X 0,Y 594.289,Z 460.029,A -85,B 0,C 180,E1 -993.728,E2 -993.728} C_VEL
LIN {X 0,Y 594.241,Z 456.132,A -85,B 0,C 180,E1 -994.747,E2 -994.747} C_VEL
LIN {X 0,Y 594.299,Z 451.108,A -85,B 0,C 180,E1 -995.767,E2 -995.767} C_VEL
LIN {X 0,Y 594.314,Z 444.798,A -85,B 0,C 180,E1 -996.79,E2 -996.79} C_VEL
LIN {X 0,Y 594.345,Z 436.886,A -85,B 0,C 180,E1 -997.814,E2 -997.814} C_VEL
LIN {X 0,Y 594.365,Z 428.82,A -85,B 0,C 180,E1 -998.669,E2 -998.669} C_VEL
LIN {X 0,Y 594.415,Z 418.968,A -85,B 0,C 180,E1 -999.526,E2 -999.526} C_VEL
LIN {X 0,Y 594.462,Z 407.947,A -85,B 0,C 180,E1 -1000.299,E2 -1000.299} C_VEL
LIN {X 0,Y 594.501,Z 395.246,A -85,B 0,C 180,E1 -1000.994,E2 -1000.994} C_VEL
LIN {X 0,Y 594.574,Z 382.872,A -85,B 0,C 180,E1 -1001.502,E2 -1001.502} C_VEL
LIN {X 0,Y 594.658,Z 370.408,A -85,B 0,C 180,E1 -1001.87,E2 -1001.87} C_VEL
LIN {X 0,Y 594.452,Z 362.063,A -85,B 0,C 180,E1 -1002.047,E2 -1002.047} C_VEL
LIN {X 0,Y 594.257,Z 360.68,A -85,B 0,C 180,E1 -1002.094,E2 -1002.094} C_VEL
LIN {X 0,Y 594.271,Z 353.352,A -85,B 0,C 180,E1 -1005.079,E2 -1005.079} C_VEL
LIN {X 0,Y 594.286,Z 348.217,A -85,B 0,C 180,E1 -1007.194,E2 -1007.194} C_VEL
LIN {X 0,Y 594.28,Z 343.082,A -85,B 0,C 180,E1 -1009.335,E2 -1009.335} C_VEL
LIN {X 0,Y 594.283,Z 337.946,A -85,B 0,C 180,E1 -1011.504,E2 -1011.504} C_VEL
LIN {X 0,Y 594.336,Z 331.099,A -85,B 0,C 180,E1 -1014.446,E2 -1014.446} C_VEL
LIN {X 0,Y 594.314,Z 325.963,A -85,B 0,C 180,E1 -1016.7,E2 -1016.7} C_VEL
LIN {X 0,Y 594.353,Z 319.244,A -85,B 0,C 180,E1 -1019.775,E2 -1019.775} C_VEL
LIN {X 0,Y 594.38,Z 313.925,A -85,B 0,C 180,E1 -1022.144,E2 -1022.144} C_VEL
LIN {X 0,Y 594.423,Z 308.118,A -85,B 0,C 180,E1 -1024.574,E2 -1024.574} C_VEL
LIN {X 0,Y 594.366,Z 306.762,A -85,B 0,C 180,E1 -1025.14,E2 -1025.14} C_VEL
LIN {X 0,Y 594.381,Z 306.76,A -85,B 0,C 180,E1 -1027.938,E2 -1027.938} C_VEL
LIN {X 0,Y 594.356,Z 306.759,A -85,B 0,C 180,E1 -1030.819,E2 -1030.819} C_VEL
LIN {X 0,Y 594.344,Z 306.762,A -85,B 0,C 180,E1 -1033.837,E2 -1033.837} C_VEL
LIN {X 0,Y 594.358,Z 306.763,A -85,B 0,C 180,E1 -1036.699,E2 -1036.699} C_VEL
LIN {X 0,Y 594.376,Z 306.756,A -85,B 0,C 180,E1 -1039.433,E2 -1039.433} C_VEL
LIN {X 0,Y 594.375,Z 306.761,A -85,B 0,C 180,E1 -1042.389,E2 -1042.389} C_VEL
LIN {X 0,Y 594.337,Z 306.761,A -85,B 0,C 180,E1 -1044.674,E2 -1044.674} C_VEL
LIN {X 0,Y 594.357,Z 306.761,A -85,B 0,C 180,E1 -1047.087,E2 -1047.087} C_VEL
LIN {X 0,Y 594.363,Z 306.759,A -85,B 0,C 180,E1 -1049.67,E2 -1049.67} C_VEL
LIN {X 0,Y 594.387,Z 306.761,A -85,B 0,C 180,E1 -1052.539,E2 -1052.539} C_VEL
LIN {X 0,Y 594.371,Z 306.759,A -85,B 0,C 180,E1 -1054.806,E2 -1054.806} C_VEL
LIN {X 0,Y 594.385,Z 306.755,A -85,B 0,C 180,E1 -1057.253,E2 -1057.253} C_VEL
LIN {X 0,Y 594.358,Z 306.761,A -85,B 0,C 180,E1 -1059.945,E2 -1059.945} C_VEL
LIN {X 0,Y 594.36,Z 306.761,A -85,B 0,C 180,E1 -1062.805,E2 -1062.805} C_VEL
LIN {X 0,Y 594.363,Z 306.757,A -85,B 0,C 180,E1 -1065.825,E2 -1065.825} C_VEL
LIN {X 0,Y 594.432,Z 306.75,A -85,B 0,C 180,E1 -1068.891,E2 -1068.891} C_VEL
LIN {X 0,Y 594.403,Z 306.76,A -85,B 0,C 180,E1 -1071.843,E2 -1071.843} C_VEL
LIN {X 0,Y 594.372,Z 306.756,A -85,B 0,C 180,E1 -1074.572,E2 -1074.572} C_VEL
LIN {X 0,Y 594.384,Z 306.76,A -85,B 0,C 180,E1 -1077.289,E2 -1077.289} C_VEL
LIN {X 0,Y 594.376,Z 306.756,A -85,B 0,C 180,E1 -1080,E2 -1080} C_VEL
LIN {X 0,Y 594.405,Z 306.755,A -85,B 0,C 180,E1 -1082.711,E2 -1082.711} C_VEL
LIN {X 0,Y 594.391,Z 306.756,A -85,B 0,C 180,E1 -1085.428,E2 -1085.428} C_VEL
LIN {X 0,Y 594.397,Z 306.754,A -85,B 0,C 180,E1 -1088.157,E2 -1088.157} C_VEL
LIN {X 0,Y 594.428,Z 306.758,A -85,B 0,C 180,E1 -1091.107,E2 -1091.107} C_VEL
LIN {X 0,Y 594.361,Z 306.763,A -85,B 0,C 180,E1 -1094.377,E2 -1094.377} C_VEL
LIN {X 0,Y 594.374,Z 306.756,A -85,B 0,C 180,E1 -1097.194,E2 -1097.194} C_VEL
LIN {X 0,Y 594.366,Z 306.762,A -85,B 0,C 180,E1 -1100.054,E2 -1100.054} C_VEL
LIN {X 0,Y 594.395,Z 306.757,A -85,B 0,C 180,E1 -1102.966,E2 -1102.966} C_VEL
LIN {X 0,Y 594.351,Z 306.765,A -85,B 0,C 180,E1 -1105.194,E2 -1105.194} C_VEL
LIN {X 0,Y 594.323,Z 306.763,A -85,B 0,C 180,E1 -1107.521,E2 -1107.521} C_VEL
LIN {X 0,Y 594.364,Z 306.765,A -85,B 0,C 180,E1 -1110.33,E2 -1110.33} C_VEL
LIN {X 0,Y 594.365,Z 306.757,A -85,B 0,C 180,E1 -1112.951,E2 -1112.951} C_VEL
LIN {X 0,Y 594.369,Z 306.763,A -85,B 0,C 180,E1 -1115.407,E2 -1115.407} C_VEL
LIN {X 0,Y 594.37,Z 306.757,A -85,B 0,C 180,E1 -1117.942,E2 -1117.942} C_VEL
LIN {X 0,Y 594.363,Z 306.765,A -85,B 0,C 180,E1 -1120.824,E2 -1120.824} C_VEL
LIN {X 0,Y 594.329,Z 306.762,A -85,B 0,C 180,E1 -1123.303,E2 -1123.303} C_VEL
LIN {X 0,Y 594.365,Z 306.764,A -85,B 0,C 180,E1 -1126.161,E2 -1126.161} C_VEL
LIN {X 0,Y 594.376,Z 306.76,A -85,B 0,C 180,E1 -1129.178,E2 -1129.178} C_VEL
LIN {X 0,Y 594.374,Z 306.756,A -85,B 0,C 180,E1 -1132.061,E2 -1132.061} C_VEL
LIN {X 0,Y 594.355,Z 306.781,A -85,B 0,C 180,E1 -1134.736,E2 -1134.736} C_VEL
LIN {X 0,Y 595.567,Z 311.697,A -85,B 0,C 180,E1 -1135.502,E2 -1135.502} C_VEL
LIN {X 0,Y 595.519,Z 326.517,A -85,B 0,C 180,E1 -1137.525,E2 -1137.525} C_VEL
LIN {X 0,Y 595.317,Z 347.265,A -85,B 0,C 180,E1 -1140.278,E2 -1140.278} C_VEL
LIN {X 0,Y 595.123,Z 369.495,A -85,B 0,C 180,E1 -1143.149,E2 -1143.149} C_VEL
LIN {X 0,Y 594.985,Z 391.725,A -85,B 0,C 180,E1 -1145.953,E2 -1145.953} C_VEL
LIN {X 0,Y 594.779,Z 413.797,A -85,B 0,C 180,E1 -1148.677,E2 -1148.677} C_VEL
LIN {X 0,Y 594.767,Z 420.762,A -85,B 0,C 180,E1 -1149.528,E2 -1149.528} C_VEL
LIN {X 0,Y 595.5,Z 424.6,A -85,B 0,C 180,E1 -1149.605,E2 -1149.605} C_VEL
LIN {X 0,Y 595.432,Z 444.891,A -85,B 0,C 180,E1 -1149.896,E2 -1149.896} C_VEL
LIN {X 0,Y 595.352,Z 461.721,A -85,B 0,C 180,E1 -1150.275,E2 -1150.275} C_VEL
LIN {X 0,Y 595.262,Z 477.763,A -85,B 0,C 180,E1 -1150.784,E2 -1150.784} C_VEL
LIN {X 0,Y 595.099,Z 493.119,A -85,B 0,C 180,E1 -1151.408,E2 -1151.408} C_VEL
LIN {X 0,Y 594.99,Z 508.913,A -85,B 0,C 180,E1 -1152.206,E2 -1152.206} C_VEL
LIN {X 0,Y 594.87,Z 522.936,A -85,B 0,C 180,E1 -1153.059,E2 -1153.059} C_VEL
LIN {X 0,Y 594.73,Z 536.718,A -85,B 0,C 180,E1 -1154.055,E2 -1154.055} C_VEL
LIN {X 0,Y 594.636,Z 549.029,A -85,B 0,C 180,E1 -1155.106,E2 -1155.106} C_VEL
LIN {X 0,Y 594.536,Z 560.136,A -85,B 0,C 180,E1 -1156.204,E2 -1156.204} C_VEL
LIN {X 0,Y 594.42,Z 571.708,A -85,B 0,C 180,E1 -1157.541,E2 -1157.541} C_VEL
LIN {X 0,Y 594.384,Z 580.634,A -85,B 0,C 180,E1 -1158.744,E2 -1158.744} C_VEL
LIN {X 0,Y 594.337,Z 589.296,A -85,B 0,C 180,E1 -1160.129,E2 -1160.129} C_VEL
LIN {X 0,Y 594.294,Z 596.495,A -85,B 0,C 180,E1 -1161.501,E2 -1161.501} C_VEL
LIN {X 0,Y 594.287,Z 602.475,A -85,B 0,C 180,E1 -1162.869,E2 -1162.869} C_VEL
LIN {X 0,Y 594.264,Z 608.251,A -85,B 0,C 180,E1 -1164.573,E2 -1164.573} C_VEL
LIN {X 0,Y 594.252,Z 611.636,A -85,B 0,C 180,E1 -1165.933,E2 -1165.933} C_VEL
LIN {X 0,Y 594.213,Z 614.089,A -85,B 0,C 180,E1 -1167.29,E2 -1167.29} C_VEL
LIN {X 0,Y 594.24,Z 615.478,A -85,B 0,C 180,E1 -1168.646,E2 -1168.646} C_VEL
LIN {X 0,Y 594.231,Z 616,A -85,B 0,C 180,E1 -1170.002,E2 -1170.002} C_VEL
LIN {X 0,Y 594.24,Z 615.476,A -85,B 0,C 180,E1 -1171.357,E2 -1171.357} C_VEL
LIN {X 0,Y 594.213,Z 614.084,A -85,B 0,C 180,E1 -1172.713,E2 -1172.713} C_VEL
LIN {X 0,Y 594.252,Z 611.63,A -85,B 0,C 180,E1 -1174.071,E2 -1174.071} C_VEL
LIN {X 0,Y 594.281,Z 607.18,A -85,B 0,C 180,E1 -1175.771,E2 -1175.771} C_VEL
LIN {X 0,Y 594.285,Z 602.463,A -85,B 0,C 180,E1 -1177.134,E2 -1177.134} C_VEL
LIN {X 0,Y 594.318,Z 594.85,A -85,B 0,C 180,E1 -1178.845,E2 -1178.845} C_VEL
LIN {X 0,Y 594.354,Z 586.237,A -85,B 0,C 180,E1 -1180.39,E2 -1180.39} C_VEL
LIN {X 0,Y 594.408,Z 576.958,A -85,B 0,C 180,E1 -1181.77,E2 -1181.77} C_VEL
LIN {X 0,Y 594.469,Z 567.41,A -85,B 0,C 180,E1 -1182.982,E2 -1182.982} C_VEL
LIN {X 0,Y 594.543,Z 555.936,A -85,B 0,C 180,E1 -1184.233,E2 -1184.233} C_VEL
LIN {X 0,Y 594.682,Z 544.127,A -85,B 0,C 180,E1 -1185.334,E2 -1185.334} C_VEL
LIN {X 0,Y 594.81,Z 530.868,A -85,B 0,C 180,E1 -1186.387,E2 -1186.387} C_VEL
LIN {X 0,Y 594.93,Z 516.408,A -85,B 0,C 180,E1 -1187.356,E2 -1187.356} C_VEL
LIN {X 0,Y 595.039,Z 502.236,A -85,B 0,C 180,E1 -1188.152,E2 -1188.152} C_VEL
LIN {X 0,Y 595.197,Z 487.114,A -85,B 0,C 180,E1 -1188.854,E2 -1188.854} C_VEL
LIN {X 0,Y 595.272,Z 471.309,A -85,B 0,C 180,E1 -1189.44,E2 -1189.44} C_VEL
LIN {X 0,Y 595.386,Z 455.295,A -85,B 0,C 180,E1 -1189.885,E2 -1189.885} C_VEL
LIN {X 0,Y 595.464,Z 439.347,A -85,B 0,C 180,E1 -1190.197,E2 -1190.197} C_VEL
LIN {X 0,Y 595.371,Z 423.675,A -85,B 0,C 180,E1 -1190.411,E2 -1190.411} C_VEL
LIN {X 0,Y 594.777,Z 420.595,A -85,B 0,C 180,E1 -1190.492,E2 -1190.492} C_VEL
LIN {X 0,Y 594.919,Z 397.624,A -85,B 0,C 180,E1 -1193.314,E2 -1193.314} C_VEL
LIN {X 0,Y 595.09,Z 376.876,A -85,B 0,C 180,E1 -1195.912,E2 -1195.912} C_VEL
LIN {X 0,Y 595.243,Z 354.646,A -85,B 0,C 180,E1 -1198.761,E2 -1198.761} C_VEL
LIN {X 0,Y 595.431,Z 335.38,A -85,B 0,C 180,E1 -1201.289,E2 -1201.289} C_VEL
LIN {X 0,Y 595.628,Z 315.229,A -85,B 0,C 180,E1 -1204.007,E2 -1204.007} C_VEL
LIN {X 0,Y 595.283,Z 310.186,A -85,B 0,C 180,E1 -1204.727,E2 -1204.727} C_VEL
LIN {X 0,Y 594.374,Z 306.762,A -85,B 0,C 180,E1 -1205.267,E2 -1205.267} C_VEL
LIN {X 0,Y 594.377,Z 306.762,A -85,B 0,C 180,E1 -1207.943,E2 -1207.943} C_VEL
LIN {X 0,Y 594.375,Z 306.761,A -85,B 0,C 180,E1 -1210.822,E2 -1210.822} C_VEL
LIN {X 0,Y 594.364,Z 306.761,A -85,B 0,C 180,E1 -1213.839,E2 -1213.839} C_VEL
LIN {X 0,Y 594.348,Z 306.763,A -85,B 0,C 180,E1 -1216.699,E2 -1216.699} C_VEL
LIN {X 0,Y 594.374,Z 306.76,A -85,B 0,C 180,E1 -1219.434,E2 -1219.434} C_VEL
LIN {X 0,Y 594.388,Z 306.758,A -85,B 0,C 180,E1 -1222.393,E2 -1222.393} C_VEL
LIN {X 0,Y 594.403,Z 306.803,A -85,B 0,C 180,E1 -1225.422,E2 -1225.422} C_VEL
LIN {X 0,Y 594.385,Z 313.478,A -85,B 0,C 180,E1 -1227.854,E2 -1227.854} C_VEL
LIN {X 0,Y 594.42,Z 319.248,A -85,B 0,C 180,E1 -1230.226,E2 -1230.226} C_VEL
LIN {X 0,Y 594.346,Z 324.046,A -85,B 0,C 180,E1 -1232.482,E2 -1232.482} C_VEL
LIN {X 0,Y 594.32,Z 329.176,A -85,B 0,C 180,E1 -1234.805,E2 -1234.805} C_VEL
LIN {X 0,Y 594.306,Z 336.019,A -85,B 0,C 180,E1 -1237.765,E2 -1237.765} C_VEL
LIN {X 0,Y 594.252,Z 341.152,A -85,B 0,C 180,E1 -1239.942,E2 -1239.942} C_VEL
LIN {X 0,Y 594.235,Z 346.284,A -85,B 0,C 180,E1 -1242.092,E2 -1242.092} C_VEL
LIN {X 0,Y 594.257,Z 353.128,A -85,B 0,C 180,E1 -1244.919,E2 -1244.919} C_VEL
LIN {X 0,Y 594.25,Z 360.72,A -85,B 0,C 180,E1 -1248.012,E2 -1248.012} C_VEL
LIN {X 0,Y 594.662,Z 365.294,A -85,B 0,C 180,E1 -1248.107,E2 -1248.107} C_VEL
LIN {X 0,Y 594.617,Z 377.445,A -85,B 0,C 180,E1 -1248.409,E2 -1248.409} C_VEL
LIN {X 0,Y 594.563,Z 389.578,A -85,B 0,C 180,E1 -1248.844,E2 -1248.844} C_VEL
LIN {X 0,Y 594.467,Z 401.962,A -85,B 0,C 180,E1 -1249.441,E2 -1249.441} C_VEL
LIN {X 0,Y 594.442,Z 413.091,A -85,B 0,C 180,E1 -1250.129,E2 -1250.129} C_VEL
LIN {X 0,Y 594.406,Z 422.103,A -85,B 0,C 180,E1 -1250.816,E2 -1250.816} C_VEL
LIN {X 0,Y 594.373,Z 431.362,A -85,B 0,C 180,E1 -1251.672,E2 -1251.672} C_VEL
LIN {X 0,Y 594.317,Z 440.335,A -85,B 0,C 180,E1 -1252.697,E2 -1252.697} C_VEL
LIN {X 0,Y 594.285,Z 446.861,A -85,B 0,C 180,E1 -1253.613,E2 -1253.613} C_VEL
LIN {X 0,Y 594.289,Z 452.442,A -85,B 0,C 180,E1 -1254.572,E2 -1254.572} C_VEL
LIN {X 0,Y 594.27,Z 457.184,A -85,B 0,C 180,E1 -1255.592,E2 -1255.592} C_VEL
LIN {X 0,Y 594.268,Z 460.818,A -85,B 0,C 180,E1 -1256.61,E2 -1256.61} C_VEL
LIN {X 0,Y 594.225,Z 462.695,A -85,B 0,C 180,E1 -1257.289,E2 -1257.289} C_VEL
LIN {X 0,Y 594.24,Z 464.128,A -85,B 0,C 180,E1 -1257.967,E2 -1257.967} C_VEL
LIN {X 0,Y 594.24,Z 465.753,A -85,B 0,C 180,E1 -1259.323,E2 -1259.323} C_VEL
LIN {X 0,Y 594.236,Z 465.996,A -85,B 0,C 180,E1 -1260,E2 -1260} C_VEL
LIN {X 0,Y 594.239,Z 465.815,A -85,B 0,C 180,E1 -1260.678,E2 -1260.678} C_VEL
LIN {X 0,Y 594.239,Z 464.275,A -85,B 0,C 180,E1 -1262.034,E2 -1262.034} C_VEL
LIN {X 0,Y 594.227,Z 462.915,A -85,B 0,C 180,E1 -1262.712,E2 -1262.712} C_VEL
LIN {X 0,Y 594.289,Z 460.037,A -85,B 0,C 180,E1 -1263.73,E2 -1263.73} C_VEL
LIN {X 0,Y 594.242,Z 456.137,A -85,B 0,C 180,E1 -1264.749,E2 -1264.749} C_VEL
LIN {X 0,Y 594.299,Z 451.107,A -85,B 0,C 180,E1 -1265.769,E2 -1265.769} C_VEL
LIN {X 0,Y 594.317,Z 444.785,A -85,B 0,C 180,E1 -1266.792,E2 -1266.792} C_VEL
LIN {X 0,Y 594.347,Z 436.868,A -85,B 0,C 180,E1 -1267.816,E2 -1267.816} C_VEL
LIN {X 0,Y 594.382,Z 427.021,A -85,B 0,C 180,E1 -1268.842,E2 -1268.842} C_VEL
LIN {X 0,Y 594.423,Z 416.698,A -85,B 0,C 180,E1 -1269.7,E2 -1269.7} C_VEL
LIN {X 0,Y 594.479,Z 405.074,A -85,B 0,C 180,E1 -1270.473,E2 -1270.473} C_VEL
LIN {X 0,Y 594.565,Z 393.246,A -85,B 0,C 180,E1 -1271.086,E2 -1271.086} C_VEL
LIN {X 0,Y 594.609,Z 380.223,A -85,B 0,C 180,E1 -1271.592,E2 -1271.592} C_VEL
LIN {X 0,Y 594.649,Z 372.728,A -85,B 0,C 180,E1 -1271.814,E2 -1271.814} C_VEL
LIN {X 0,Y 593.895,Z 368.894,A -85,B 0,C 180,E1 -1271.953,E2 -1271.953} C_VEL
LIN {X 0,Y 591.562,Z 364.567,A -85,B 0,C 180,E1 -1272.22,E2 -1272.22} C_VEL
LIN {X 0,Y 588.953,Z 361.179,A -85,B 0,C 180,E1 -1272.576,E2 -1272.576} C_VEL
LIN {X 0,Y 587.518,Z 359.289,A -85,B 0,C 180,E1 -1272.909,E2 -1272.909} C_VEL
LIN {X 0,Y 587.16,Z 358.441,A -85,B 0,C 180,E1 -1273.161,E2 -1273.161} C_VEL
LIN {X 0,Y 587.148,Z 351.633,A -85,B 0,C 180,E1 -1275.98,E2 -1275.98} C_VEL
LIN {X 0,Y 587.216,Z 344.435,A -85,B 0,C 180,E1 -1279.002,E2 -1279.002} C_VEL
LIN {X 0,Y 587.21,Z 337.939,A -85,B 0,C 180,E1 -1281.779,E2 -1281.779} C_VEL
LIN {X 0,Y 587.248,Z 331.561,A -85,B 0,C 180,E1 -1284.556,E2 -1284.556} C_VEL
LIN {X 0,Y 587.283,Z 326.061,A -85,B 0,C 180,E1 -1287.049,E2 -1287.049} C_VEL
LIN {X 0,Y 587.328,Z 320.959,A -85,B 0,C 180,E1 -1289.381,E2 -1289.381} C_VEL
LIN {X 0,Y 587.363,Z 315.589,A -85,B 0,C 180,E1 -1291.837,E2 -1291.837} C_VEL
LIN {X 0,Y 587.366,Z 310.129,A -85,B 0,C 180,E1 -1294.349,E2 -1294.349} C_VEL
LIN {X 0,Y 587.361,Z 307.636,A -85,B 0,C 180,E1 -1295.545,E2 -1295.545} C_VEL
LIN {X 0,Y 587.327,Z 307.639,A -85,B 0,C 180,E1 -1298.48,E2 -1298.48} C_VEL
LIN {X 0,Y 587.342,Z 307.638,A -85,B 0,C 180,E1 -1301.157,E2 -1301.157} C_VEL
LIN {X 0,Y 587.326,Z 307.64,A -85,B 0,C 180,E1 -1304.112,E2 -1304.112} C_VEL
LIN {X 0,Y 587.299,Z 307.642,A -85,B 0,C 180,E1 -1306.991,E2 -1306.991} C_VEL
LIN {X 0,Y 587.315,Z 307.64,A -85,B 0,C 180,E1 -1309.745,E2 -1309.745} C_VEL
LIN {X 0,Y 587.351,Z 307.636,A -85,B 0,C 180,E1 -1312.392,E2 -1312.392} C_VEL
LIN {X 0,Y 587.341,Z 307.792,A -85,B 0,C 180,E1 -1314.944,E2 -1314.944} C_VEL
LIN {X 0,Y 587.403,Z 312.536,A -85,B 0,C 180,E1 -1316.879,E2 -1316.879} C_VEL
LIN {X 0,Y 587.343,Z 318.405,A -85,B 0,C 180,E1 -1319.49,E2 -1319.49} C_VEL
LIN {X 0,Y 587.29,Z 324.569,A -85,B 0,C 180,E1 -1322.319,E2 -1322.319} C_VEL
LIN {X 0,Y 587.257,Z 329.178,A -85,B 0,C 180,E1 -1324.479,E2 -1324.479} C_VEL
LIN {X 0,Y 587.258,Z 336.017,A -85,B 0,C 180,E1 -1327.482,E2 -1327.482} C_VEL
LIN {X 0,Y 587.201,Z 341.149,A -85,B 0,C 180,E1 -1329.689,E2 -1329.689} C_VEL
LIN {X 0,Y 587.191,Z 346.282,A -85,B 0,C 180,E1 -1331.868,E2 -1331.868} C_VEL
LIN {X 0,Y 587.174,Z 351.414,A -85,B 0,C 180,E1 -1334.019,E2 -1334.019} C_VEL
LIN {X 0,Y 587.195,Z 356.547,A -85,B 0,C 180,E1 -1336.149,E2 -1336.149} C_VEL
LIN {X 0,Y 587.161,Z 360.718,A -85,B 0,C 180,E1 -1337.864,E2 -1337.864} C_VEL
LIN {X 0,Y 587.74,Z 366.395,A -85,B 0,C 180,E1 -1337.985,E2 -1337.985} C_VEL
LIN {X 0,Y 587.631,Z 378.874,A -85,B 0,C 180,E1 -1338.315,E2 -1338.315} C_VEL
LIN {X 0,Y 587.556,Z 390.831,A -85,B 0,C 180,E1 -1338.766,E2 -1338.766} C_VEL
LIN {X 0,Y 587.505,Z 401.907,A -85,B 0,C 180,E1 -1339.313,E2 -1339.313} C_VEL
LIN {X 0,Y 587.461,Z 413.055,A -85,B 0,C 180,E1 -1340.009,E2 -1340.009} C_VEL
LIN {X 0,Y 587.352,Z 424.084,A -85,B 0,C 180,E1 -1340.876,E2 -1340.876} C_VEL
LIN {X 0,Y 587.303,Z 432.979,A -85,B 0,C 180,E1 -1341.742,E2 -1341.742} C_VEL
LIN {X 0,Y 587.261,Z 440.323,A -85,B 0,C 180,E1 -1342.607,E2 -1342.607} C_VEL
LIN {X 0,Y 587.198,Z 447.414,A -85,B 0,C 180,E1 -1343.624,E2 -1343.624} C_VEL
LIN {X 0,Y 587.211,Z 452.421,A -85,B 0,C 180,E1 -1344.504,E2 -1344.504} C_VEL
LIN {X 0,Y 587.188,Z 457.158,A -85,B 0,C 180,E1 -1345.536,E2 -1345.536} C_VEL
LIN {X 0,Y 587.194,Z 460.8,A -85,B 0,C 180,E1 -1346.568,E2 -1346.568} C_VEL
LIN {X 0,Y 587.132,Z 462.687,A -85,B 0,C 180,E1 -1347.254,E2 -1347.254} C_VEL
LIN {X 0,Y 587.141,Z 464.131,A -85,B 0,C 180,E1 -1347.94,E2 -1347.94} C_VEL
LIN {X 0,Y 587.14,Z 465.754,A -85,B 0,C 180,E1 -1349.313,E2 -1349.313} C_VEL
LIN {X 0,Y 587.137,Z 465.995,A -85,B 0,C 180,E1 -1349.998,E2 -1349.998} C_VEL
LIN {X 0,Y 587.148,Z 465.235,A -85,B 0,C 180,E1 -1351.37,E2 -1351.37} C_VEL
LIN {X 0,Y 587.141,Z 464.28,A -85,B 0,C 180,E1 -1352.056,E2 -1352.056} C_VEL
LIN {X 0,Y 587.132,Z 462.894,A -85,B 0,C 180,E1 -1352.743,E2 -1352.743} C_VEL
LIN {X 0,Y 587.213,Z 460.021,A -85,B 0,C 180,E1 -1353.773,E2 -1353.773} C_VEL
LIN {X 0,Y 587.146,Z 456.124,A -85,B 0,C 180,E1 -1354.805,E2 -1354.805} C_VEL
LIN {X 0,Y 587.229,Z 451.101,A -85,B 0,C 180,E1 -1355.837,E2 -1355.837} C_VEL
LIN {X 0,Y 587.228,Z 444.794,A -85,B 0,C 180,E1 -1356.872,E2 -1356.872} C_VEL
LIN {X 0,Y 587.287,Z 436.882,A -85,B 0,C 180,E1 -1357.908,E2 -1357.908} C_VEL
LIN {X 0,Y 587.324,Z 428.814,A -85,B 0,C 180,E1 -1358.774,E2 -1358.774} C_VEL
LIN {X 0,Y 587.387,Z 418.947,A -85,B 0,C 180,E1 -1359.641,E2 -1359.641} C_VEL
LIN {X 0,Y 587.452,Z 409.27,A -85,B 0,C 180,E1 -1360.336,E2 -1360.336} C_VEL
LIN {X 0,Y 587.519,Z 397.134,A -85,B 0,C 180,E1 -1361.032,E2 -1361.032} C_VEL
LIN {X 0,Y 587.607,Z 384.005,A -85,B 0,C 180,E1 -1361.6,E2 -1361.6} C_VEL
LIN {X 0,Y 587.7,Z 372.097,A -85,B 0,C 180,E1 -1361.968,E2 -1361.968} C_VEL
LIN {X 0,Y 587.5,Z 362.784,A -85,B 0,C 180,E1 -1362.178,E2 -1362.178} C_VEL
LIN {X 0,Y 587.156,Z 360.732,A -85,B 0,C 180,E1 -1362.221,E2 -1362.221} C_VEL
LIN {X 0,Y 587.202,Z 355.062,A -85,B 0,C 180,E1 -1364.555,E2 -1364.555} C_VEL
LIN {X 0,Y 587.209,Z 348.215,A -85,B 0,C 180,E1 -1367.408,E2 -1367.408} C_VEL
LIN {X 0,Y 587.206,Z 343.08,A -85,B 0,C 180,E1 -1369.578,E2 -1369.578} C_VEL
LIN {X 0,Y 587.257,Z 336.233,A -85,B 0,C 180,E1 -1372.515,E2 -1372.515} C_VEL
LIN {X 0,Y 587.254,Z 329.385,A -85,B 0,C 180,E1 -1375.518,E2 -1375.518} C_VEL
LIN {X 0,Y 587.278,Z 324.496,A -85,B 0,C 180,E1 -1377.819,E2 -1377.819} C_VEL
LIN {X 0,Y 587.337,Z 318.623,A -85,B 0,C 180,E1 -1380.509,E2 -1380.509} C_VEL
LIN {X 0,Y 587.407,Z 312.118,A -85,B 0,C 180,E1 -1383.389,E2 -1383.389} C_VEL
LIN {X 0,Y 587.328,Z 307.638,A -85,B 0,C 180,E1 -1385.227,E2 -1385.227} C_VEL
LIN {X 0,Y 587.334,Z 307.637,A -85,B 0,C 180,E1 -1387.837,E2 -1387.837} C_VEL
LIN {X 0,Y 587.302,Z 307.641,A -85,B 0,C 180,E1 -1390.252,E2 -1390.252} C_VEL
LIN {X 0,Y 587.282,Z 307.643,A -85,B 0,C 180,E1 -1393.114,E2 -1393.114} C_VEL
LIN {X 0,Y 587.306,Z 307.637,A -85,B 0,C 180,E1 -1396.048,E2 -1396.048} C_VEL
LIN {X 0,Y 587.35,Z 307.635,A -85,B 0,C 180,E1 -1398.92,E2 -1398.92} C_VEL
LIN {X 0,Y 587.32,Z 307.635,A -85,B 0,C 180,E1 -1401.52,E2 -1401.52} C_VEL
LIN {X 0,Y 587.33,Z 307.639,A -85,B 0,C 180,E1 -1404.102,E2 -1404.102} C_VEL
LIN {X 0,Y 587.316,Z 307.637,A -85,B 0,C 180,E1 -1406.887,E2 -1406.887} C_VEL
LIN {X 0,Y 587.31,Z 307.636,A -85,B 0,C 180,E1 -1409.828,E2 -1409.828} C_VEL
LIN {X 0,Y 587.33,Z 307.637,A -85,B 0,C 180,E1 -1412.305,E2 -1412.305} C_VEL
LIN {X 0,Y 587.329,Z 307.641,A -85,B 0,C 180,E1 -1414.483,E2 -1414.483} C_VEL
LIN {X 0,Y 587.35,Z 307.633,A -85,B 0,C 180,E1 -1417.486,E2 -1417.486} C_VEL
LIN {X 0,Y 587.321,Z 307.634,A -85,B 0,C 180,E1 -1420.424,E2 -1420.424} C_VEL
LIN {X 0,Y 587.322,Z 307.64,A -85,B 0,C 180,E1 -1423.31,E2 -1423.31} C_VEL
LIN {X 0,Y 587.341,Z 307.633,A -85,B 0,C 180,E1 -1426.154,E2 -1426.154} C_VEL
LIN {X 0,Y 587.387,Z 307.627,A -85,B 0,C 180,E1 -1428.963,E2 -1428.963} C_VEL
LIN {X 0,Y 587.356,Z 307.636,A -85,B 0,C 180,E1 -1431.744,E2 -1431.744} C_VEL
LIN {X 0,Y 587.337,Z 307.632,A -85,B 0,C 180,E1 -1434.507,E2 -1434.507} C_VEL
LIN {X 0,Y 587.35,Z 307.637,A -85,B 0,C 180,E1 -1437.256,E2 -1437.256} C_VEL
LIN {X 0,Y 587.346,Z 307.632,A -85,B 0,C 180,E1 -1440,E2 -1440} C_VEL
LIN {X 0,Y 587.369,Z 307.631,A -85,B 0,C 180,E1 -1442.743,E2 -1442.743} C_VEL
LIN {X 0,Y 587.357,Z 307.633,A -85,B 0,C 180,E1 -1445.493,E2 -1445.493} C_VEL
LIN {X 0,Y 587.35,Z 307.632,A -85,B 0,C 180,E1 -1448.255,E2 -1448.255} C_VEL
LIN {X 0,Y 587.385,Z 307.634,A -85,B 0,C 180,E1 -1451.166,E2 -1451.166} C_VEL
LIN {X 0,Y 587.313,Z 307.644,A -85,B 0,C 180,E1 -1454.554,E2 -1454.554} C_VEL
LIN {X 0,Y 587.341,Z 307.633,A -85,B 0,C 180,E1 -1457.406,E2 -1457.406} C_VEL
LIN {X 0,Y 587.331,Z 307.638,A -85,B 0,C 180,E1 -1459.575,E2 -1459.575} C_VEL
LIN {X 0,Y 587.348,Z 307.631,A -85,B 0,C 180,E1 -1462.513,E2 -1462.513} C_VEL
LIN {X 0,Y 587.305,Z 307.639,A -85,B 0,C 180,E1 -1465.518,E2 -1465.518} C_VEL
LIN {X 0,Y 587.31,Z 307.636,A -85,B 0,C 180,E1 -1467.819,E2 -1467.819} C_VEL
LIN {X 0,Y 587.32,Z 307.64,A -85,B 0,C 180,E1 -1470.512,E2 -1470.512} C_VEL
LIN {X 0,Y 587.324,Z 307.635,A -85,B 0,C 180,E1 -1473.114,E2 -1473.114} C_VEL
LIN {X 0,Y 587.341,Z 307.636,A -85,B 0,C 180,E1 -1475.896,E2 -1475.896} C_VEL
LIN {X 0,Y 587.317,Z 307.637,A -85,B 0,C 180,E1 -1478.48,E2 -1478.48} C_VEL
LIN {X 0,Y 587.314,Z 307.638,A -85,B 0,C 180,E1 -1481.159,E2 -1481.159} C_VEL
LIN {X 0,Y 587.297,Z 307.643,A -85,B 0,C 180,E1 -1484.114,E2 -1484.114} C_VEL
LIN {X 0,Y 587.306,Z 307.638,A -85,B 0,C 180,E1 -1486.996,E2 -1486.996} C_VEL
LIN {X 0,Y 587.315,Z 307.642,A -85,B 0,C 180,E1 -1489.749,E2 -1489.749} C_VEL
LIN {X 0,Y 587.333,Z 307.633,A -85,B 0,C 180,E1 -1492.395,E2 -1492.395} C_VEL
LIN {X 0,Y 587.328,Z 307.783,A -85,B 0,C 180,E1 -1494.393,E2 -1494.393} C_VEL
LIN {X 0,Y 588.989,Z 314.25,A -85,B 0,C 180,E1 -1495.419,E2 -1495.419} C_VEL
LIN {X 0,Y 588.847,Z 331.537,A -85,B 0,C 180,E1 -1497.798,E2 -1497.798} C_VEL
LIN {X 0,Y 588.565,Z 353.193,A -85,B 0,C 180,E1 -1500.69,E2 -1500.69} C_VEL
LIN {X 0,Y 588.32,Z 373.922,A -85,B 0,C 180,E1 -1503.387,E2 -1503.387} C_VEL
LIN {X 0,Y 588.112,Z 396.171,A -85,B 0,C 180,E1 -1506.217,E2 -1506.217} C_VEL
LIN {X 0,Y 587.876,Z 420.763,A -85,B 0,C 180,E1 -1509.277,E2 -1509.277} C_VEL
LIN {X 0,Y 588.85,Z 426.389,A -85,B 0,C 180,E1 -1509.387,E2 -1509.387} C_VEL
LIN {X 0,Y 588.783,Z 446.031,A -85,B 0,C 180,E1 -1509.681,E2 -1509.681} C_VEL
LIN {X 0,Y 588.67,Z 461.72,A -85,B 0,C 180,E1 -1510.042,E2 -1510.042} C_VEL
LIN {X 0,Y 588.54,Z 477.994,A -85,B 0,C 180,E1 -1510.563,E2 -1510.563} C_VEL
LIN {X 0,Y 588.347,Z 493.121,A -85,B 0,C 180,E1 -1511.187,E2 -1511.187} C_VEL
LIN {X 0,Y 588.161,Z 508.914,A -85,B 0,C 180,E1 -1511.992,E2 -1511.992} C_VEL
LIN {X 0,Y 587.999,Z 523.713,A -85,B 0,C 180,E1 -1512.909,E2 -1512.909} C_VEL
LIN {X 0,Y 587.84,Z 536.719,A -85,B 0,C 180,E1 -1513.863,E2 -1513.863} C_VEL
LIN {X 0,Y 587.675,Z 549.03,A -85,B 0,C 180,E1 -1514.926,E2 -1514.926} C_VEL
LIN {X 0,Y 587.575,Z 559.642,A -85,B 0,C 180,E1 -1515.984,E2 -1515.984} C_VEL
LIN {X 0,Y 587.425,Z 570.348,A -85,B 0,C 180,E1 -1517.215,E2 -1517.215} C_VEL
LIN {X 0,Y 587.349,Z 580.69,A -85,B 0,C 180,E1 -1518.615,E2 -1518.615} C_VEL
LIN {X 0,Y 587.289,Z 589.297,A -85,B 0,C 180,E1 -1520.009,E2 -1520.009} C_VEL
LIN {X 0,Y 587.238,Z 596.496,A -85,B 0,C 180,E1 -1521.398,E2 -1521.398} C_VEL
LIN {X 0,Y 587.21,Z 602.475,A -85,B 0,C 180,E1 -1522.782,E2 -1522.782} C_VEL
LIN {X 0,Y 587.187,Z 608.251,A -85,B 0,C 180,E1 -1524.507,E2 -1524.507} C_VEL
LIN {X 0,Y 587.167,Z 611.637,A -85,B 0,C 180,E1 -1525.883,E2 -1525.883} C_VEL
LIN {X 0,Y 587.119,Z 614.089,A -85,B 0,C 180,E1 -1527.257,E2 -1527.257} C_VEL
LIN {X 0,Y 587.14,Z 615.479,A -85,B 0,C 180,E1 -1528.63,E2 -1528.63} C_VEL
LIN {X 0,Y 587.132,Z 616,A -85,B 0,C 180,E1 -1530.002,E2 -1530.002} C_VEL
LIN {X 0,Y 587.14,Z 615.477,A -85,B 0,C 180,E1 -1531.373,E2 -1531.373} C_VEL
LIN {X 0,Y 587.119,Z 614.084,A -85,B 0,C 180,E1 -1532.746,E2 -1532.746} C_VEL
LIN {X 0,Y 587.167,Z 611.63,A -85,B 0,C 180,E1 -1534.12,E2 -1534.12} C_VEL
LIN {X 0,Y 587.189,Z 607.18,A -85,B 0,C 180,E1 -1535.841,E2 -1535.841} C_VEL
LIN {X 0,Y 587.209,Z 602.462,A -85,B 0,C 180,E1 -1537.221,E2 -1537.221} C_VEL
LIN {X 0,Y 587.246,Z 594.85,A -85,B 0,C 180,E1 -1538.952,E2 -1538.952} C_VEL
LIN {X 0,Y 587.302,Z 586.238,A -85,B 0,C 180,E1 -1540.516,E2 -1540.516} C_VEL
LIN {X 0,Y 587.368,Z 576.959,A -85,B 0,C 180,E1 -1541.913,E2 -1541.913} C_VEL
LIN {X 0,Y 587.449,Z 567.41,A -85,B 0,C 180,E1 -1543.14,E2 -1543.14} C_VEL
LIN {X 0,Y 587.565,Z 556.62,A -85,B 0,C 180,E1 -1544.337,E2 -1544.337} C_VEL
LIN {X 0,Y 587.721,Z 544.127,A -85,B 0,C 180,E1 -1545.521,E2 -1545.521} C_VEL
LIN {X 0,Y 587.911,Z 529.691,A -85,B 0,C 180,E1 -1546.674,E2 -1546.674} C_VEL
LIN {X 0,Y 588.091,Z 514.993,A -85,B 0,C 180,E1 -1547.654,E2 -1547.654} C_VEL
LIN {X 0,Y 588.254,Z 500.49,A -85,B 0,C 180,E1 -1548.459,E2 -1548.459} C_VEL
LIN {X 0,Y 588.449,Z 484.332,A -85,B 0,C 180,E1 -1549.191,E2 -1549.191} C_VEL
LIN {X 0,Y 588.612,Z 468.439,A -85,B 0,C 180,E1 -1549.759,E2 -1549.759} C_VEL
LIN {X 0,Y 588.727,Z 452.551,A -85,B 0,C 180,E1 -1550.187,E2 -1550.187} C_VEL
LIN {X 0,Y 588.83,Z 436.335,A -85,B 0,C 180,E1 -1550.48,E2 -1550.48} C_VEL
LIN {X 0,Y 588.69,Z 424.772,A -85,B 0,C 180,E1 -1550.639,E2 -1550.639} C_VEL
LIN {X 0,Y 587.869,Z 420.595,A -85,B 0,C 180,E1 -1550.744,E2 -1550.744} C_VEL
LIN {X 0,Y 588.1,Z 397.624,A -85,B 0,C 180,E1 -1553.6,E2 -1553.6} C_VEL
LIN {X 0,Y 588.309,Z 375.822,A -85,B 0,C 180,E1 -1556.369,E2 -1556.369} C_VEL
LIN {X 0,Y 588.577,Z 352.906,A -85,B 0,C 180,E1 -1559.347,E2 -1559.347} C_VEL
LIN {X 0,Y 588.826,Z 332.532,A -85,B 0,C 180,E1 -1562.067,E2 -1562.067} C_VEL
LIN {X 0,Y 589.044,Z 315.393,A -85,B 0,C 180,E1 -1564.417,E2 -1564.417} C_VEL
LIN {X 0,Y 588.463,Z 311.668,A -85,B 0,C 180,E1 -1564.979,E2 -1564.979} C_VEL
LIN {X 0,Y 587.307,Z 307.642,A -85,B 0,C 180,E1 -1565.638,E2 -1565.638} C_VEL
LIN {X 0,Y 587.324,Z 307.639,A -85,B 0,C 180,E1 -1568.481,E2 -1568.481} C_VEL
LIN {X 0,Y 587.337,Z 307.637,A -85,B 0,C 180,E1 -1571.158,E2 -1571.158} C_VEL
LIN {X 0,Y 587.316,Z 307.639,A -85,B 0,C 180,E1 -1574.113,E2 -1574.113} C_VEL
LIN {X 0,Y 587.295,Z 307.643,A -85,B 0,C 180,E1 -1576.992,E2 -1576.992} C_VEL
LIN {X 0,Y 587.316,Z 307.64,A -85,B 0,C 180,E1 -1579.746,E2 -1579.746} C_VEL
LIN {X 0,Y 587.343,Z 307.636,A -85,B 0,C 180,E1 -1582.392,E2 -1582.392} C_VEL
LIN {X 0,Y 587.369,Z 307.7,A -85,B 0,C 180,E1 -1585.38,E2 -1585.38} C_VEL
LIN {X 0,Y 587.348,Z 313.378,A -85,B 0,C 180,E1 -1587.422,E2 -1587.422} C_VEL
LIN {X 0,Y 587.37,Z 319.282,A -85,B 0,C 180,E1 -1589.832,E2 -1589.832} C_VEL
LIN {X 0,Y 587.376,Z 322.938,A -85,B 0,C 180,E1 -1591.406,E2 -1591.406} C_VEL
LIN {X 0,Y 587.284,Z 327.888,A -85,B 0,C 180,E1 -1593.835,E2 -1593.835} C_VEL
LIN {X 0,Y 587.234,Z 332.599,A -85,B 0,C 180,E1 -1595.989,E2 -1595.989} C_VEL
LIN {X 0,Y 587.214,Z 337.732,A -85,B 0,C 180,E1 -1598.222,E2 -1598.222} C_VEL
LIN {X 0,Y 587.235,Z 344.575,A -85,B 0,C 180,E1 -1601.148,E2 -1601.148} C_VEL
LIN {X 0,Y 587.144,Z 351.418,A -85,B 0,C 180,E1 -1604.02,E2 -1604.02} C_VEL
LIN {X 0,Y 587.16,Z 356.551,A -85,B 0,C 180,E1 -1606.15,E2 -1606.15} C_VEL
LIN {X 0,Y 587.144,Z 360.722,A -85,B 0,C 180,E1 -1607.865,E2 -1607.865} C_VEL
LIN {X 0,Y 587.711,Z 366.464,A -85,B 0,C 180,E1 -1607.986,E2 -1607.986} C_VEL
LIN {X 0,Y 587.635,Z 378.937,A -85,B 0,C 180,E1 -1608.316,E2 -1608.316} C_VEL
LIN {X 0,Y 587.6,Z 391.5,A -85,B 0,C 180,E1 -1608.794,E2 -1608.794} C_VEL
LIN {X 0,Y 587.488,Z 403.54,A -85,B 0,C 180,E1 -1609.402,E2 -1609.402} C_VEL
LIN {X 0,Y 587.424,Z 414.326,A -85,B 0,C 180,E1 -1610.097,E2 -1610.097} C_VEL
LIN {X 0,Y 587.357,Z 424.1,A -85,B 0,C 180,E1 -1610.878,E2 -1610.878} C_VEL
LIN {X 0,Y 587.302,Z 432.993,A -85,B 0,C 180,E1 -1611.744,E2 -1611.744} C_VEL
LIN {X 0,Y 587.234,Z 441.678,A -85,B 0,C 180,E1 -1612.781,E2 -1612.781} C_VEL
LIN {X 0,Y 587.214,Z 448.605,A -85,B 0,C 180,E1 -1613.817,E2 -1613.817} C_VEL
LIN {X 0,Y 587.168,Z 454.156,A -85,B 0,C 180,E1 -1614.85,E2 -1614.85} C_VEL
LIN {X 0,Y 587.182,Z 458.517,A -85,B 0,C 180,E1 -1615.882,E2 -1615.882} C_VEL
LIN {X 0,Y 587.194,Z 460.82,A -85,B 0,C 180,E1 -1616.569,E2 -1616.569} C_VEL
LIN {X 0,Y 587.132,Z 462.697,A -85,B 0,C 180,E1 -1617.256,E2 -1617.256} C_VEL
LIN {X 0,Y 587.139,Z 464.128,A -85,B 0,C 180,E1 -1617.942,E2 -1617.942} C_VEL
LIN {X 0,Y 587.14,Z 465.754,A -85,B 0,C 180,E1 -1619.314,E2 -1619.314} C_VEL
LIN {X 0,Y 587.137,Z 465.996,A -85,B 0,C 180,E1 -1620,E2 -1620} C_VEL
LIN {X 0,Y 587.14,Z 465.815,A -85,B 0,C 180,E1 -1620.686,E2 -1620.686} C_VEL
LIN {X 0,Y 587.138,Z 464.274,A -85,B 0,C 180,E1 -1622.058,E2 -1622.058} C_VEL
LIN {X 0,Y 587.133,Z 462.914,A -85,B 0,C 180,E1 -1622.745,E2 -1622.745} C_VEL
LIN {X 0,Y 587.213,Z 460.035,A -85,B 0,C 180,E1 -1623.775,E2 -1623.775} C_VEL
LIN {X 0,Y 587.147,Z 456.135,A -85,B 0,C 180,E1 -1624.807,E2 -1624.807} C_VEL
LIN {X 0,Y 587.229,Z 451.104,A -85,B 0,C 180,E1 -1625.839,E2 -1625.839} C_VEL
LIN {X 0,Y 587.231,Z 444.781,A -85,B 0,C 180,E1 -1626.874,E2 -1626.874} C_VEL
LIN {X 0,Y 587.288,Z 436.864,A -85,B 0,C 180,E1 -1627.91,E2 -1627.91} C_VEL
LIN {X 0,Y 587.344,Z 427.015,A -85,B 0,C 180,E1 -1628.949,E2 -1628.949} C_VEL
LIN {X 0,Y 587.407,Z 416.692,A -85,B 0,C 180,E1 -1629.817,E2 -1629.817} C_VEL
LIN {X 0,Y 587.489,Z 405.064,A -85,B 0,C 180,E1 -1630.599,E2 -1630.599} C_VEL
LIN {X 0,Y 587.587,Z 394.175,A -85,B 0,C 180,E1 -1631.177,E2 -1631.177} C_VEL
LIN {X 0,Y 587.634,Z 381.463,A -85,B 0,C 180,E1 -1631.689,E2 -1631.689} C_VEL
LIN {X 0,Y 587.694,Z 368.478,A -85,B 0,C 180,E1 -1632.058,E2 -1632.058} C_VEL
LIN {X 0,Y 587.511,Z 363.135,A -85,B 0,C 180,E1 -1632.172,E2 -1632.172} C_VEL
LIN {X 0,Y 587.147,Z 360.726,A -85,B 0,C 180,E1 -1632.223,E2 -1632.223} C_VEL
LIN {X 0,Y 587.16,Z 358.441,A -85,B 0,C 180,E1 -1633.161,E2 -1633.161} C_VEL
LIN {X 0,Y 586.471,Z 357.127,A -85,B 0,C 180,E1 -1633.719,E2 -1633.719} C_VEL
LIN {X 0,Y 583.588,Z 355.11,A -85,B 0,C 180,E1 -1634.627,E2 -1634.627} C_VEL
LIN {X 0,Y 581.173,Z 353.514,A -85,B 0,C 180,E1 -1635.357,E2 -1635.357} C_VEL
LIN {X 0,Y 580.152,Z 352.243,A -85,B 0,C 180,E1 -1635.92,E2 -1635.92} C_VEL
LIN {X 0,Y 580.076,Z 351.797,A -85,B 0,C 180,E1 -1636.111,E2 -1636.111} C_VEL
LIN {X 0,Y 580.129,Z 344.765,A -85,B 0,C 180,E1 -1639.101,E2 -1639.101} C_VEL
LIN {X 0,Y 580.15,Z 337.937,A -85,B 0,C 180,E1 -1642.058,E2 -1642.058} C_VEL
LIN {X 0,Y 580.204,Z 331.981,A -85,B 0,C 180,E1 -1644.704,E2 -1644.704} C_VEL
LIN {X 0,Y 580.239,Z 326.188,A -85,B 0,C 180,E1 -1647.405,E2 -1647.405} C_VEL
LIN {X 0,Y 580.283,Z 320.992,A -85,B 0,C 180,E1 -1649.773,E2 -1649.773} C_VEL
LIN {X 0,Y 580.311,Z 315.754,A -85,B 0,C 180,E1 -1652.2,E2 -1652.2} C_VEL
LIN {X 0,Y 580.339,Z 310.367,A -85,B 0,C 180,E1 -1654.693,E2 -1654.693} C_VEL
LIN {X 0,Y 580.322,Z 308.513,A -85,B 0,C 180,E1 -1655.624,E2 -1655.624} C_VEL
LIN {X 0,Y 580.291,Z 308.515,A -85,B 0,C 180,E1 -1658.146,E2 -1658.146} C_VEL
LIN {X 0,Y 580.304,Z 308.513,A -85,B 0,C 180,E1 -1660.843,E2 -1660.843} C_VEL
LIN {X 0,Y 580.276,Z 308.517,A -85,B 0,C 180,E1 -1663.659,E2 -1663.659} C_VEL
LIN {X 0,Y 580.244,Z 308.523,A -85,B 0,C 180,E1 -1666.613,E2 -1666.613} C_VEL
LIN {X 0,Y 580.304,Z 308.516,A -85,B 0,C 180,E1 -1669.156,E2 -1669.156} C_VEL
LIN {X 0,Y 580.294,Z 308.516,A -85,B 0,C 180,E1 -1671.927,E2 -1671.927} C_VEL
LIN {X 0,Y 580.287,Z 308.611,A -85,B 0,C 180,E1 -1674.826,E2 -1674.826} C_VEL
LIN {X 0,Y 580.379,Z 313.903,A -85,B 0,C 180,E1 -1676.98,E2 -1676.98} C_VEL
LIN {X 0,Y 580.344,Z 319.346,A -85,B 0,C 180,E1 -1679.427,E2 -1679.427} C_VEL
LIN {X 0,Y 580.267,Z 325.204,A -85,B 0,C 180,E1 -1682.148,E2 -1682.148} C_VEL
LIN {X 0,Y 580.208,Z 331.057,A -85,B 0,C 180,E1 -1684.914,E2 -1684.914} C_VEL
LIN {X 0,Y 580.18,Z 336.019,A -85,B 0,C 180,E1 -1687.192,E2 -1687.192} C_VEL
LIN {X 0,Y 580.141,Z 341.151,A -85,B 0,C 180,E1 -1689.431,E2 -1689.431} C_VEL
LIN {X 0,Y 580.134,Z 346.283,A -85,B 0,C 180,E1 -1691.639,E2 -1691.639} C_VEL
LIN {X 0,Y 580.105,Z 351.416,A -85,B 0,C 180,E1 -1693.819,E2 -1693.819} C_VEL
LIN {X 0,Y 580.139,Z 356.549,A -85,B 0,C 180,E1 -1695.977,E2 -1695.977} C_VEL
LIN {X 0,Y 580.089,Z 360.943,A -85,B 0,C 180,E1 -1697.725,E2 -1697.725} C_VEL
LIN {X 0,Y 580.814,Z 366.426,A -85,B 0,C 180,E1 -1697.84,E2 -1697.84} C_VEL
LIN {X 0,Y 580.694,Z 378.77,A -85,B 0,C 180,E1 -1698.17,E2 -1698.17} C_VEL
LIN {X 0,Y 580.575,Z 390.689,A -85,B 0,C 180,E1 -1698.623,E2 -1698.623} C_VEL
LIN {X 0,Y 580.523,Z 401.905,A -85,B 0,C 180,E1 -1699.183,E2 -1699.183} C_VEL
LIN {X 0,Y 580.46,Z 411.782,A -85,B 0,C 180,E1 -1699.799,E2 -1699.799} C_VEL
LIN {X 0,Y 580.353,Z 422.086,A -85,B 0,C 180,E1 -1700.589,E2 -1700.589} C_VEL
LIN {X 0,Y 580.292,Z 431.359,A -85,B 0,C 180,E1 -1701.467,E2 -1701.467} C_VEL
LIN {X 0,Y 580.201,Z 440.32,A -85,B 0,C 180,E1 -1702.516,E2 -1702.516} C_VEL
LIN {X 0,Y 580.171,Z 446.346,A -85,B 0,C 180,E1 -1703.377,E2 -1703.377} C_VEL
LIN {X 0,Y 580.14,Z 452.416,A -85,B 0,C 180,E1 -1704.437,E2 -1704.437} C_VEL
LIN {X 0,Y 580.108,Z 457.154,A -85,B 0,C 180,E1 -1705.482,E2 -1705.482} C_VEL
LIN {X 0,Y 580.123,Z 460.798,A -85,B 0,C 180,E1 -1706.526,E2 -1706.526} C_VEL
LIN {X 0,Y 580.043,Z 462.681,A -85,B 0,C 180,E1 -1707.22,E2 -1707.22} C_VEL
LIN {X 0,Y 580.04,Z 464.132,A -85,B 0,C 180,E1 -1707.915,E2 -1707.915} C_VEL
LIN {X 0,Y 580.041,Z 465.755,A -85,B 0,C 180,E1 -1709.304,E2 -1709.304} C_VEL
LIN {X 0,Y 580.038,Z 465.996,A -85,B 0,C 180,E1 -1709.998,E2 -1709.998} C_VEL
LIN {X 0,Y 580.047,Z 465.234,A -85,B 0,C 180,E1 -1711.387,E2 -1711.387} C_VEL
LIN {X 0,Y 580.04,Z 464.281,A -85,B 0,C 180,E1 -1712.081,E2 -1712.081} C_VEL
LIN {X 0,Y 580.123,Z 461.082,A -85,B 0,C 180,E1 -1713.471,E2 -1713.471} C_VEL
LIN {X 0,Y 580.108,Z 457.535,A -85,B 0,C 180,E1 -1714.515,E2 -1714.515} C_VEL
LIN {X 0,Y 580.137,Z 452.892,A -85,B 0,C 180,E1 -1715.56,E2 -1715.56} C_VEL
LIN {X 0,Y 580.131,Z 447.124,A -85,B 0,C 180,E1 -1716.589,E2 -1716.589} C_VEL
LIN {X 0,Y 580.219,Z 439.694,A -85,B 0,C 180,E1 -1717.655,E2 -1717.655} C_VEL
LIN {X 0,Y 580.258,Z 430.581,A -85,B 0,C 180,E1 -1718.706,E2 -1718.706} C_VEL
LIN {X 0,Y 580.359,Z 421.093,A -85,B 0,C 180,E1 -1719.583,E2 -1719.583} C_VEL
LIN {X 0,Y 580.433,Z 410.557,A -85,B 0,C 180,E1 -1720.374,E2 -1720.374} C_VEL
LIN {X 0,Y 580.505,Z 400.41,A -85,B 0,C 180,E1 -1720.991,E2 -1720.991} C_VEL
LIN {X 0,Y 580.619,Z 389.22,A -85,B 0,C 180,E1 -1721.532,E2 -1721.532} C_VEL
LIN {X 0,Y 580.75,Z 376.104,A -85,B 0,C 180,E1 -1722.003,E2 -1722.003} C_VEL
LIN {X 0,Y 580.679,Z 364.394,A -85,B 0,C 180,E1 -1722.293,E2 -1722.293} C_VEL
LIN {X 0,Y 580.09,Z 360.73,A -85,B 0,C 180,E1 -1722.372,E2 -1722.372} C_VEL
LIN {X 0,Y 580.118,Z 355.061,A -85,B 0,C 180,E1 -1724.737,E2 -1724.737} C_VEL
LIN {X 0,Y 580.138,Z 348.214,A -85,B 0,C 180,E1 -1727.627,E2 -1727.627} C_VEL
LIN {X 0,Y 580.133,Z 343.079,A -85,B 0,C 180,E1 -1729.826,E2 -1729.826} C_VEL
LIN {X 0,Y 580.18,Z 337.943,A -85,B 0,C 180,E1 -1732.054,E2 -1732.054} C_VEL
LIN {X 0,Y 580.214,Z 332.084,A -85,B 0,C 180,E1 -1734.706,E2 -1734.706} C_VEL
LIN {X 0,Y 580.24,Z 326.389,A -85,B 0,C 180,E1 -1737.402,E2 -1737.402} C_VEL
LIN {X 0,Y 580.304,Z 321.284,A -85,B 0,C 180,E1 -1739.769,E2 -1739.769} C_VEL
LIN {X 0,Y 580.343,Z 315.993,A -85,B 0,C 180,E1 -1742.195,E2 -1742.195} C_VEL
LIN {X 0,Y 580.381,Z 310.119,A -85,B 0,C 180,E1 -1744.687,E2 -1744.687} C_VEL
LIN {X 0,Y 580.315,Z 308.512,A -85,B 0,C 180,E1 -1745.327,E2 -1745.327} C_VEL
LIN {X 0,Y 580.279,Z 308.52,A -85,B 0,C 180,E1 -1748.144,E2 -1748.144} C_VEL
LIN {X 0,Y 580.283,Z 308.512,A -85,B 0,C 180,E1 -1750.841,E2 -1750.841} C_VEL
LIN {X 0,Y 580.252,Z 308.52,A -85,B 0,C 180,E1 -1753.657,E2 -1753.657} C_VEL
LIN {X 0,Y 580.269,Z 308.517,A -85,B 0,C 180,E1 -1756.606,E2 -1756.606} C_VEL
LIN {X 0,Y 580.306,Z 308.51,A -85,B 0,C 180,E1 -1759.157,E2 -1759.157} C_VEL
LIN {X 0,Y 580.276,Z 308.517,A -85,B 0,C 180,E1 -1761.925,E2 -1761.925} C_VEL
LIN {X 0,Y 580.268,Z 308.514,A -85,B 0,C 180,E1 -1764.453,E2 -1764.453} C_VEL
LIN {X 0,Y 580.268,Z 308.515,A -85,B 0,C 180,E1 -1766.973,E2 -1766.973} C_VEL
LIN {X 0,Y 580.273,Z 308.516,A -85,B 0,C 180,E1 -1769.423,E2 -1769.423} C_VEL
LIN {X 0,Y 580.3,Z 308.511,A -85,B 0,C 180,E1 -1772.135,E2 -1772.135} C_VEL
LIN {X 0,Y 580.293,Z 308.512,A -85,B 0,C 180,E1 -1774.919,E2 -1774.919} C_VEL
LIN {X 0,Y 580.33,Z 308.505,A -85,B 0,C 180,E1 -1777.199,E2 -1777.199} C_VEL
LIN {X 0,Y 580.286,Z 308.512,A -85,B 0,C 180,E1 -1780.177,E2 -1780.177} C_VEL
LIN {X 0,Y 580.282,Z 308.519,A -85,B 0,C 180,E1 -1783.101,E2 -1783.101} C_VEL
LIN {X 0,Y 580.304,Z 308.508,A -85,B 0,C 180,E1 -1785.982,E2 -1785.982} C_VEL
LIN {X 0,Y 580.365,Z 308.503,A -85,B 0,C 180,E1 -1788.828,E2 -1788.828} C_VEL
LIN {X 0,Y 580.319,Z 308.51,A -85,B 0,C 180,E1 -1791.644,E2 -1791.644} C_VEL
LIN {X 0,Y 580.303,Z 308.508,A -85,B 0,C 180,E1 -1794.44,E2 -1794.44} C_VEL
LIN {X 0,Y 580.315,Z 308.514,A -85,B 0,C 180,E1 -1797.223,E2 -1797.223} C_VEL
LIN {X 0,Y 580.316,Z 308.507,A -85,B 0,C 180,E1 -1800,E2 -1800} C_VEL
LIN {X 0,Y 580.333,Z 308.507,A -85,B 0,C 180,E1 -1802.776,E2 -1802.776} C_VEL
LIN {X 0,Y 580.323,Z 308.51,A -85,B 0,C 180,E1 -1805.559,E2 -1805.559} C_VEL
LIN {X 0,Y 580.314,Z 308.508,A -85,B 0,C 180,E1 -1808.356,E2 -1808.356} C_VEL
LIN {X 0,Y 580.337,Z 308.511,A -85,B 0,C 180,E1 -1811.224,E2 -1811.224} C_VEL
LIN {X 0,Y 580.281,Z 308.516,A -85,B 0,C 180,E1 -1814.336,E2 -1814.336} C_VEL
LIN {X 0,Y 580.318,Z 308.508,A -85,B 0,C 180,E1 -1816.925,E2 -1816.925} C_VEL
LIN {X 0,Y 580.292,Z 308.518,A -85,B 0,C 180,E1 -1819.822,E2 -1819.822} C_VEL
LIN {X 0,Y 580.328,Z 308.507,A -85,B 0,C 180,E1 -1822.801,E2 -1822.801} C_VEL
LIN {X 0,Y 580.28,Z 308.52,A -85,B 0,C 180,E1 -1825.081,E2 -1825.081} C_VEL
LIN {X 0,Y 580.272,Z 308.515,A -85,B 0,C 180,E1 -1828.187,E2 -1828.187} C_VEL
LIN {X 0,Y 580.27,Z 308.516,A -85,B 0,C 180,E1 -1830.698,E2 -1830.698} C_VEL
LIN {X 0,Y 580.289,Z 308.513,A -85,B 0,C 180,E1 -1833.319,E2 -1833.319} C_VEL
LIN {X 0,Y 580.31,Z 308.513,A -85,B 0,C 180,E1 -1835.77,E2 -1835.77} C_VEL
LIN {X 0,Y 580.27,Z 308.513,A -85,B 0,C 180,E1 -1838.147,E2 -1838.147} C_VEL
LIN {X 0,Y 580.281,Z 308.518,A -85,B 0,C 180,E1 -1840.845,E2 -1840.845} C_VEL
LIN {X 0,Y 580.247,Z 308.516,A -85,B 0,C 180,E1 -1843.661,E2 -1843.661} C_VEL
LIN {X 0,Y 580.268,Z 308.516,A -85,B 0,C 180,E1 -1846.61,E2 -1846.61} C_VEL
LIN {X 0,Y 580.305,Z 308.513,A -85,B 0,C 180,E1 -1849.16,E2 -1849.16} C_VEL
LIN {X 0,Y 580.277,Z 308.511,A -85,B 0,C 180,E1 -1851.928,E2 -1851.928} C_VEL
LIN {X 0,Y 580.272,Z 308.655,A -85,B 0,C 180,E1 -1854.018,E2 -1854.018} C_VEL
LIN {X 0,Y 582.218,Z 315.722,A -85,B 0,C 180,E1 -1855.168,E2 -1855.168} C_VEL
LIN {X 0,Y 582.43,Z 320.589,A -85,B 0,C 180,E1 -1855.871,E2 -1855.871} C_VEL
LIN {X 0,Y 582.036,Z 342.947,A -85,B 0,C 180,E1 -1858.943,E2 -1858.943} C_VEL
LIN {X 0,Y 581.675,Z 365.049,A -85,B 0,C 180,E1 -1861.89,E2 -1861.89} C_VEL
LIN {X 0,Y 581.376,Z 385.797,A -85,B 0,C 180,E1 -1864.589,E2 -1864.589} C_VEL
LIN {X 0,Y 581.161,Z 405.254,A -85,B 0,C 180,E1 -1867.072,E2 -1867.072} C_VEL
LIN {X 0,Y 580.983,Z 420.717,A -85,B 0,C 180,E1 -1869.014,E2 -1869.014} C_VEL
LIN {X 0,Y 582.19,Z 426.389,A -85,B 0,C 180,E1 -1869.141,E2 -1869.141} C_VEL
LIN {X 0,Y 582.133,Z 446.031,A -85,B 0,C 180,E1 -1869.439,E2 -1869.439} C_VEL
LIN {X 0,Y 581.995,Z 461.72,A -85,B 0,C 180,E1 -1869.803,E2 -1869.803} C_VEL
LIN {X 0,Y 581.813,Z 477.95,A -85,B 0,C 180,E1 -1870.328,E2 -1870.328} C_VEL
LIN {X 0,Y 581.574,Z 493.122,A -85,B 0,C 180,E1 -1870.959,E2 -1870.959} C_VEL
LIN {X 0,Y 581.351,Z 508.916,A -85,B 0,C 180,E1 -1871.774,E2 -1871.774} C_VEL
LIN {X 0,Y 581.143,Z 522.985,A -85,B 0,C 180,E1 -1872.65,E2 -1872.65} C_VEL
LIN {X 0,Y 580.945,Z 536.72,A -85,B 0,C 180,E1 -1873.666,E2 -1873.666} C_VEL
LIN {X 0,Y 580.71,Z 549.03,A -85,B 0,C 180,E1 -1874.74,E2 -1874.74} C_VEL
LIN {X 0,Y 580.594,Z 559.961,A -85,B 0,C 180,E1 -1875.847,E2 -1875.847} C_VEL
LIN {X 0,Y 580.41,Z 570.349,A -85,B 0,C 180,E1 -1877.057,E2 -1877.057} C_VEL
LIN {X 0,Y 580.313,Z 580.69,A -85,B 0,C 180,E1 -1878.476,E2 -1878.476} C_VEL
LIN {X 0,Y 580.218,Z 589.298,A -85,B 0,C 180,E1 -1879.886,E2 -1879.886} C_VEL
LIN {X 0,Y 580.163,Z 596.497,A -85,B 0,C 180,E1 -1881.293,E2 -1881.293} C_VEL
LIN {X 0,Y 580.121,Z 602.475,A -85,B 0,C 180,E1 -1882.694,E2 -1882.694} C_VEL
LIN {X 0,Y 580.111,Z 608.25,A -85,B 0,C 180,E1 -1884.44,E2 -1884.44} C_VEL
LIN {X 0,Y 580.085,Z 611.637,A -85,B 0,C 180,E1 -1885.833,E2 -1885.833} C_VEL
LIN {X 0,Y 580.031,Z 614.089,A -85,B 0,C 180,E1 -1887.224,E2 -1887.224} C_VEL
LIN {X 0,Y 580.04,Z 615.479,A -85,B 0,C 180,E1 -1888.613,E2 -1888.613} C_VEL
LIN {X 0,Y 580.033,Z 616,A -85,B 0,C 180,E1 -1890.002,E2 -1890.002} C_VEL
LIN {X 0,Y 580.04,Z 615.477,A -85,B 0,C 180,E1 -1891.39,E2 -1891.39} C_VEL
LIN {X 0,Y 580.031,Z 614.084,A -85,B 0,C 180,E1 -1892.78,E2 -1892.78} C_VEL
LIN {X 0,Y 580.085,Z 611.63,A -85,B 0,C 180,E1 -1894.17,E2 -1894.17} C_VEL
LIN {X 0,Y 580.1,Z 607.181,A -85,B 0,C 180,E1 -1895.912,E2 -1895.912} C_VEL
LIN {X 0,Y 580.12,Z 602.462,A -85,B 0,C 180,E1 -1897.31,E2 -1897.31} C_VEL
LIN {X 0,Y 580.157,Z 594.85,A -85,B 0,C 180,E1 -1899.062,E2 -1899.062} C_VEL
LIN {X 0,Y 580.241,Z 586.239,A -85,B 0,C 180,E1 -1900.646,E2 -1900.646} C_VEL
LIN {X 0,Y 580.337,Z 576.959,A -85,B 0,C 180,E1 -1902.059,E2 -1902.059} C_VEL
LIN {X 0,Y 580.441,Z 567.411,A -85,B 0,C 180,E1 -1903.302,E2 -1903.302} C_VEL
LIN {X 0,Y 580.604,Z 555.917,A -85,B 0,C 180,E1 -1904.584,E2 -1904.584} C_VEL
LIN {X 0,Y 580.815,Z 544.127,A -85,B 0,C 180,E1 -1905.71,E2 -1905.71} C_VEL
LIN {X 0,Y 581.012,Z 530.866,A -85,B 0,C 180,E1 -1906.787,E2 -1906.787} C_VEL
LIN {X 0,Y 581.25,Z 516.411,A -85,B 0,C 180,E1 -1907.778,E2 -1907.778} C_VEL
LIN {X 0,Y 581.445,Z 502.239,A -85,B 0,C 180,E1 -1908.592,E2 -1908.592} C_VEL
LIN {X 0,Y 581.707,Z 487.06,A -85,B 0,C 180,E1 -1909.311,E2 -1909.311} C_VEL
LIN {X 0,Y 581.872,Z 471.308,A -85,B 0,C 180,E1 -1909.906,E2 -1909.906} C_VEL
LIN {X 0,Y 582.043,Z 455.297,A -85,B 0,C 180,E1 -1910.36,E2 -1910.36} C_VEL
LIN {X 0,Y 582.179,Z 439.347,A -85,B 0,C 180,E1 -1910.679,E2 -1910.679} C_VEL
LIN {X 0,Y 582.111,Z 426.111,A -85,B 0,C 180,E1 -1910.866,E2 -1910.866} C_VEL
LIN {X 0,Y 580.97,Z 420.596,A -85,B 0,C 180,E1 -1911.002,E2 -1911.002} C_VEL
LIN {X 0,Y 581.267,Z 397.624,A -85,B 0,C 180,E1 -1913.895,E2 -1913.895} C_VEL
LIN {X 0,Y 581.552,Z 375.543,A -85,B 0,C 180,E1 -1916.736,E2 -1916.736} C_VEL
LIN {X 0,Y 581.876,Z 353.164,A -85,B 0,C 180,E1 -1919.684,E2 -1919.684} C_VEL
LIN {X 0,Y 582.156,Z 333.676,A -85,B 0,C 180,E1 -1922.322,E2 -1922.322} C_VEL
LIN {X 0,Y 582.447,Z 317.596,A -85,B 0,C 180,E1 -1924.551,E2 -1924.551} C_VEL
LIN {X 0,Y 581.54,Z 313.059,A -85,B 0,C 180,E1 -1925.259,E2 -1925.259} C_VEL
LIN {X 0,Y 580.266,Z 308.521,A -85,B 0,C 180,E1 -1926.007,E2 -1926.007} C_VEL
LIN {X 0,Y 580.287,Z 308.516,A -85,B 0,C 180,E1 -1928.148,E2 -1928.148} C_VEL
LIN {X 0,Y 580.301,Z 308.514,A -85,B 0,C 180,E1 -1930.844,E2 -1930.844} C_VEL
LIN {X 0,Y 580.273,Z 308.517,A -85,B 0,C 180,E1 -1933.66,E2 -1933.66} C_VEL
LIN {X 0,Y 580.243,Z 308.52,A -85,B 0,C 180,E1 -1936.614,E2 -1936.614} C_VEL
LIN {X 0,Y 580.302,Z 308.514,A -85,B 0,C 180,E1 -1939.157,E2 -1939.157} C_VEL
LIN {X 0,Y 580.288,Z 308.516,A -85,B 0,C 180,E1 -1941.928,E2 -1941.928} C_VEL
LIN {X 0,Y 580.294,Z 308.516,A -85,B 0,C 180,E1 -1944.881,E2 -1944.881} C_VEL
LIN {X 0,Y 580.335,Z 308.6,A -85,B 0,C 180,E1 -1945.307,E2 -1945.307} C_VEL
LIN {X 0,Y 580.342,Z 315.452,A -85,B 0,C 180,E1 -1947.802,E2 -1947.802} C_VEL
LIN {X 0,Y 580.348,Z 321.27,A -85,B 0,C 180,E1 -1950.231,E2 -1950.231} C_VEL
LIN {X 0,Y 580.293,Z 326.413,A -85,B 0,C 180,E1 -1952.599,E2 -1952.599} C_VEL
LIN {X 0,Y 580.231,Z 331.21,A -85,B 0,C 180,E1 -1954.917,E2 -1954.917} C_VEL
LIN {X 0,Y 580.183,Z 336.022,A -85,B 0,C 180,E1 -1957.193,E2 -1957.193} C_VEL
LIN {X 0,Y 580.134,Z 341.155,A -85,B 0,C 180,E1 -1959.432,E2 -1959.432} C_VEL
LIN {X 0,Y 580.108,Z 346.287,A -85,B 0,C 180,E1 -1961.64,E2 -1961.64} C_VEL
LIN {X 0,Y 580.087,Z 353.131,A -85,B 0,C 180,E1 -1964.542,E2 -1964.542} C_VEL
LIN {X 0,Y 580.067,Z 359.975,A -85,B 0,C 180,E1 -1967.404,E2 -1967.404} C_VEL
LIN {X 0,Y 580.065,Z 360.723,A -85,B 0,C 180,E1 -1967.715,E2 -1967.715} C_VEL
LIN {X 0,Y 580.769,Z 366.493,A -85,B 0,C 180,E1 -1967.841,E2 -1967.841} C_VEL
LIN {X 0,Y 580.708,Z 378.867,A -85,B 0,C 180,E1 -1968.172,E2 -1968.172} C_VEL
LIN {X 0,Y 580.645,Z 391.136,A -85,B 0,C 180,E1 -1968.641,E2 -1968.641} C_VEL
LIN {X 0,Y 580.495,Z 403.552,A -85,B 0,C 180,E1 -1969.272,E2 -1969.272} C_VEL
LIN {X 0,Y 580.426,Z 414.332,A -85,B 0,C 180,E1 -1969.976,E2 -1969.976} C_VEL
LIN {X 0,Y 580.333,Z 424.106,A -85,B 0,C 180,E1 -1970.767,E2 -1970.767} C_VEL
LIN {X 0,Y 580.265,Z 432.999,A -85,B 0,C 180,E1 -1971.643,E2 -1971.643} C_VEL
LIN {X 0,Y 580.176,Z 441.682,A -85,B 0,C 180,E1 -1972.693,E2 -1972.693} C_VEL
LIN {X 0,Y 580.137,Z 448.609,A -85,B 0,C 180,E1 -1973.741,E2 -1973.741} C_VEL
LIN {X 0,Y 580.086,Z 454.159,A -85,B 0,C 180,E1 -1974.787,E2 -1974.787} C_VEL
LIN {X 0,Y 580.105,Z 458.518,A -85,B 0,C 180,E1 -1975.832,E2 -1975.832} C_VEL
LIN {X 0,Y 580.123,Z 460.822,A -85,B 0,C 180,E1 -1976.528,E2 -1976.528} C_VEL
LIN {X 0,Y 580.043,Z 462.699,A -85,B 0,C 180,E1 -1977.222,E2 -1977.222} C_VEL
LIN {X 0,Y 580.038,Z 464.128,A -85,B 0,C 180,E1 -1977.917,E2 -1977.917} C_VEL
LIN {X 0,Y 580.041,Z 465.755,A -85,B 0,C 180,E1 -1979.306,E2 -1979.306} C_VEL
LIN {X 0,Y 580.038,Z 465.996,A -85,B 0,C 180,E1 -1980,E2 -1980} C_VEL
LIN {X 0,Y 580.04,Z 465.815,A -85,B 0,C 180,E1 -1980.695,E2 -1980.695} C_VEL
LIN {X 0,Y 580.037,Z 464.273,A -85,B 0,C 180,E1 -1982.083,E2 -1982.083} C_VEL
LIN {X 0,Y 580.044,Z 462.913,A -85,B 0,C 180,E1 -1982.778,E2 -1982.778} C_VEL
LIN {X 0,Y 580.11,Z 460.034,A -85,B 0,C 180,E1 -1983.821,E2 -1983.821} C_VEL
LIN {X 0,Y 580.054,Z 456.133,A -85,B 0,C 180,E1 -1984.866,E2 -1984.866} C_VEL
LIN {X 0,Y 580.162,Z 451.102,A -85,B 0,C 180,E1 -1985.91,E2 -1985.91} C_VEL
LIN {X 0,Y 580.159,Z 444.777,A -85,B 0,C 180,E1 -1986.958,E2 -1986.958} C_VEL
LIN {X 0,Y 580.242,Z 436.858,A -85,B 0,C 180,E1 -1988.007,E2 -1988.007} C_VEL
LIN {X 0,Y 580.309,Z 427.009,A -85,B 0,C 180,E1 -1989.059,E2 -1989.059} C_VEL
LIN {X 0,Y 580.405,Z 416.686,A -85,B 0,C 180,E1 -1989.936,E2 -1989.936} C_VEL
LIN {X 0,Y 580.507,Z 405.053,A -85,B 0,C 180,E1 -1990.728,E2 -1990.728} C_VEL
LIN {X 0,Y 580.614,Z 393.496,A -85,B 0,C 180,E1 -1991.343,E2 -1991.343} C_VEL
LIN {X 0,Y 580.686,Z 381.617,A -85,B 0,C 180,E1 -1991.825,E2 -1991.825} C_VEL
LIN {X 0,Y 580.773,Z 368.455,A -85,B 0,C 180,E1 -1992.204,E2 -1992.204} C_VEL
LIN {X 0,Y 580.422,Z 363.106,A -85,B 0,C 180,E1 -1992.323,E2 -1992.323} C_VEL
LIN {X 0,Y 580.085,Z 360.725,A -85,B 0,C 180,E1 -1992.374,E2 -1992.374} C_VEL
LIN {X 0,Y 580.101,Z 355.055,A -85,B 0,C 180,E1 -1994.739,E2 -1994.739} C_VEL
LIN {X 0,Y 580.076,Z 351.797,A -85,B 0,C 180,E1 -1996.111,E2 -1996.111} C_VEL
LIN {X 0,Y 579.422,Z 350.505,A -85,B 0,C 180,E1 -1996.676,E2 -1996.676} C_VEL
LIN {X 0,Y 576.549,Z 348.55,A -85,B 0,C 180,E1 -1997.596,E2 -1997.596} C_VEL
LIN {X 0,Y 574.129,Z 347.007,A -85,B 0,C 180,E1 -1998.337,E2 -1998.337} C_VEL
LIN {X 0,Y 573.116,Z 345.766,A -85,B 0,C 180,E1 -1998.908,E2 -1998.908} C_VEL
LIN {X 0,Y 573.048,Z 345.328,A -85,B 0,C 180,E1 -1999.101,E2 -1999.101} C_VEL
LIN {X 0,Y 573.08,Z 339.648,A -85,B 0,C 180,E1 -2001.587,E2 -2001.587} C_VEL
LIN {X 0,Y 573.117,Z 334.601,A -85,B 0,C 180,E1 -2003.871,E2 -2003.871} C_VEL
